LIN {X -6.399,Y 248.174,Z 120.000,A 0.000,B 0.000,C 180.000,E1 0.000} C_DIS
LIN {X -19.159,Y 247.517,Z 120.000,A 0.000,B 0.000,C 180.000,E1 0.000} C_DIS
LIN {X -31.876,Y 246.202,Z 120.000,A 0.000,B 0.000,C 180.000,E1 0.000} C_DIS
LIN {X -44.507,Y 244.235,Z 120.000,A 0.000,B 0.000,C 180.000,E1 0.000} C_DIS
LIN {X -57.020,Y 241.620,Z 120.000,A 0.000,B 0.000,C 180.000,E1 0.000} C_DIS
LIN {X -69.385,Y 238.363,Z 120.000,A 0.000,B 0.000,C 180.000,E1 0.000} C_DIS
LIN {X -81.563,Y 234.476,Z 120.000,A 0.000,B 0.000,C 180.000,E1 0.000} C_DIS
LIN {X -93.525,Y 229.967,Z 120.000,A 0.000,B 0.000,C 180.000,E1 0.000} C_DIS
LIN {X -105.240,Y 224.847,Z 120.000,A 0.000,B 0.000,C 180.000,E1 0.000} C_DIS
LIN {X -116.676,Y 219.131,Z 120.000,A 0.000,B 0.000,C 180.000,E1 0.000} C_DIS
LIN {X -127.801,Y 212.835,Z 120.000,A 0.000,B 0.000,C 180.000,E1 0.000} C_DIS
LIN {X -138.588,Y 205.972,Z 120.000,A 0.000,B 0.000,C 180.000,E1 0.000} C_DIS
LIN {X -149.007,Y 198.566,Z 120.000,A 0.000,B 0.000,C 180.000,E1 0.000} C_DIS
LIN {X -159.031,Y 190.632,Z 120.000,A 0.000,B 0.000,C 180.000,E1 0.000} C_DIS
LIN {X -168.634,Y 182.192,Z 120.000,A 0.000,B 0.000,C 180.000,E1 0.000} C_DIS
LIN {X -177.790,Y 173.268,Z 120.000,A 0.000,B 0.000,C 180.000,E1 0.000} C_DIS
LIN {X -186.475,Y 163.887,Z 120.000,A 0.000,B 0.000,C 180.000,E1 0.000} C_DIS
LIN {X -194.663,Y 154.071,Z 120.000,A 0.000,B 0.000,C 180.000,E1 0.000} C_DIS
LIN {X -202.336,Y 143.846,Z 120.000,A 0.000,B 0.000,C 180.000,E1 0.000} C_DIS
LIN {X -209.473,Y 133.237,Z 120.000,A 0.000,B 0.000,C 180.000,E1 0.000} C_DIS
LIN {X -216.056,Y 122.277,Z 120.000,A 0.000,B 0.000,C 180.000,E1 0.000} C_DIS
LIN {X -222.063,Y 110.995,Z 120.000,A 0.000,B 0.000,C 180.000,E1 0.000} C_DIS
LIN {X -227.482,Y 99.416,Z 120.000,A 0.000,B 0.000,C 180.000,E1 0.000} C_DIS
LIN {X -232.298,Y 87.573,Z 120.000,A 0.000,B 0.000,C 180.000,E1 0.000} C_DIS
LIN {X -236.498,Y 75.499,Z 120.000,A 0.000,B 0.000,C 180.000,E1 0.000} C_DIS
LIN {X -240.071,Y 63.225,Z 120.000,A 0.000,B 0.000,C 180.000,E1 0.000} C_DIS
LIN {X -243.008,Y 50.781,Z 120.000,A 0.000,B 0.000,C 180.000,E1 0.000} C_DIS
LIN {X -245.300,Y 38.205,Z 120.000,A 0.000,B 0.000,C 180.000,E1 0.000} C_DIS
LIN {X -246.940,Y 25.526,Z 120.000,A 0.000,B 0.000,C 180.000,E1 0.000} C_DIS
LIN {X -247.927,Y 12.780,Z 120.000,A 0.000,B 0.000,C 180.000,E1 0.000} C_DIS
LIN {X -248.256,Y 0.000,Z 120.000,A 0.000,B 0.000,C 180.000,E1 0.000} C_DIS
LIN {X -247.927,Y -12.780,Z 120.000,A 0.000,B 0.000,C 180.000,E1 0.000} C_DIS
LIN {X -246.940,Y -25.526,Z 120.000,A 0.000,B 0.000,C 180.000,E1 0.000} C_DIS
LIN {X -245.300,Y -38.205,Z 120.000,A 0.000,B 0.000,C 180.000,E1 0.000} C_DIS
LIN {X -243.008,Y -50.781,Z 120.000,A 0.000,B 0.000,C 180.000,E1 0.000} C_DIS
LIN {X -240.071,Y -63.225,Z 120.000,A 0.000,B 0.000,C 180.000,E1 0.000} C_DIS
LIN {X -236.498,Y -75.499,Z 120.000,A 0.000,B 0.000,C 180.000,E1 0.000} C_DIS
LIN {X -232.298,Y -87.573,Z 120.000,A 0.000,B 0.000,C 180.000,E1 0.000} C_DIS
LIN {X -227.482,Y -99.416,Z 120.000,A 0.000,B 0.000,C 180.000,E1 0.000} C_DIS
LIN {X -222.063,Y -110.995,Z 120.000,A 0.000,B 0.000,C 180.000,E1 0.000} C_DIS
LIN {X -216.056,Y -122.277,Z 120.000,A 0.000,B 0.000,C 180.000,E1 0.000} C_DIS
LIN {X -209.473,Y -133.237,Z 120.000,A 0.000,B 0.000,C 180.000,E1 0.000} C_DIS
LIN {X -202.336,Y -143.846,Z 120.000,A 0.000,B 0.000,C 180.000,E1 0.000} C_DIS
LIN {X -194.663,Y -154.071,Z 120.000,A 0.000,B 0.000,C 180.000,E1 0.000} C_DIS
LIN {X -186.475,Y -163.887,Z 120.000,A 0.000,B 0.000,C 180.000,E1 0.000} C_DIS
LIN {X -177.790,Y -173.268,Z 120.000,A 0.000,B 0.000,C 180.000,E1 0.000} C_DIS
LIN {X -168.634,Y -182.192,Z 120.000,A 0.000,B 0.000,C 180.000,E1 0.000} C_DIS
LIN {X -159.031,Y -190.632,Z 120.000,A 0.000,B 0.000,C 180.000,E1 0.000} C_DIS
LIN {X -149.007,Y -198.566,Z 120.000,A 0.000,B 0.000,C 180.000,E1 0.000} C_DIS
LIN {X -138.588,Y -205.972,Z 120.000,A 0.000,B 0.000,C 180.000,E1 0.000} C_DIS
LIN {X -127.801,Y -212.835,Z 120.000,A 0.000,B 0.000,C 180.000,E1 0.000} C_DIS
LIN {X -116.676,Y -219.131,Z 120.000,A 0.000,B 0.000,C 180.000,E1 0.000} C_DIS
LIN {X -105.240,Y -224.847,Z 120.000,A 0.000,B 0.000,C 180.000,E1 0.000} C_DIS
LIN {X -93.525,Y -229.967,Z 120.000,A 0.000,B 0.000,C 180.000,E1 0.000} C_DIS
LIN {X -81.563,Y -234.476,Z 120.000,A 0.000,B 0.000,C 180.000,E1 0.000} C_DIS
LIN {X -69.385,Y -238.363,Z 120.000,A 0.000,B 0.000,C 180.000,E1 0.000} C_DIS
LIN {X -57.020,Y -241.620,Z 120.000,A 0.000,B 0.000,C 180.000,E1 0.000} C_DIS
LIN {X -44.507,Y -244.235,Z 120.000,A 0.000,B 0.000,C 180.000,E1 0.000} C_DIS
LIN {X -31.876,Y -246.202,Z 120.000,A 0.000,B 0.000,C 180.000,E1 0.000} C_DIS
LIN {X -19.160,Y -247.517,Z 120.000,A 0.000,B 0.000,C 180.000,E1 0.000} C_DIS
LIN {X -6.393,Y -248.174,Z 120.000,A 0.000,B 0.000,C 180.000,E1 0.000} C_DIS
LIN {X 6.399,Y -248.174,Z 120.000,A 0.000,B 0.000,C 180.000,E1 0.000} C_DIS
LIN {X 19.159,Y -247.517,Z 120.000,A 0.000,B 0.000,C 180.000,E1 0.000} C_DIS
LIN {X 31.876,Y -246.202,Z 120.000,A 0.000,B 0.000,C 180.000,E1 0.000} C_DIS
LIN {X 44.507,Y -244.235,Z 120.000,A 0.000,B 0.000,C 180.000,E1 0.000} C_DIS
LIN {X 57.020,Y -241.620,Z 120.000,A 0.000,B 0.000,C 180.000,E1 0.000} C_DIS
LIN {X 69.385,Y -238.363,Z 120.000,A 0.000,B 0.000,C 180.000,E1 0.000} C_DIS
LIN {X 81.563,Y -234.476,Z 120.000,A 0.000,B 0.000,C 180.000,E1 0.000} C_DIS
LIN {X 93.525,Y -229.967,Z 120.000,A 0.000,B 0.000,C 180.000,E1 0.000} C_DIS
LIN {X 105.240,Y -224.847,Z 120.000,A 0.000,B 0.000,C 180.000,E1 0.000} C_DIS
LIN {X 116.676,Y -219.131,Z 120.000,A 0.000,B 0.000,C 180.000,E1 0.000} C_DIS
LIN {X 127.801,Y -212.835,Z 120.000,A 0.000,B 0.000,C 180.000,E1 0.000} C_DIS
LIN {X 138.588,Y -205.972,Z 120.000,A 0.000,B 0.000,C 180.000,E1 0.000} C_DIS
LIN {X 149.007,Y -198.566,Z 120.000,A 0.000,B 0.000,C 180.000,E1 0.000} C_DIS
LIN {X 159.031,Y -190.632,Z 120.000,A 0.000,B 0.000,C 180.000,E1 0.000} C_DIS
LIN {X 168.634,Y -182.192,Z 120.000,A 0.000,B 0.000,C 180.000,E1 0.000} C_DIS
LIN {X 177.790,Y -173.268,Z 120.000,A 0.000,B 0.000,C 180.000,E1 0.000} C_DIS
LIN {X 186.475,Y -163.887,Z 120.000,A 0.000,B 0.000,C 180.000,E1 0.000} C_DIS
LIN {X 194.663,Y -154.071,Z 120.000,A 0.000,B 0.000,C 180.000,E1 0.000} C_DIS
LIN {X 202.336,Y -143.846,Z 120.000,A 0.000,B 0.000,C 180.000,E1 0.000} C_DIS
LIN {X 209.473,Y -133.237,Z 120.000,A 0.000,B 0.000,C 180.000,E1 0.000} C_DIS
LIN {X 216.056,Y -122.277,Z 120.000,A 0.000,B 0.000,C 180.000,E1 0.000} C_DIS
LIN {X 222.063,Y -110.995,Z 120.000,A 0.000,B 0.000,C 180.000,E1 0.000} C_DIS
LIN {X 227.482,Y -99.416,Z 120.000,A 0.000,B 0.000,C 180.000,E1 0.000} C_DIS
LIN {X 232.298,Y -87.573,Z 120.000,A 0.000,B 0.000,C 180.000,E1 0.000} C_DIS
LIN {X 236.498,Y -75.499,Z 120.000,A 0.000,B 0.000,C 180.000,E1 0.000} C_DIS
LIN {X 240.071,Y -63.225,Z 120.000,A 0.000,B 0.000,C 180.000,E1 0.000} C_DIS
LIN {X 243.008,Y -50.781,Z 120.000,A 0.000,B 0.000,C 180.000,E1 0.000} C_DIS
LIN {X 245.300,Y -38.205,Z 120.000,A 0.000,B 0.000,C 180.000,E1 0.000} C_DIS
LIN {X 246.940,Y -25.526,Z 120.000,A 0.000,B 0.000,C 180.000,E1 0.000} C_DIS
LIN {X 247.927,Y -12.780,Z 120.000,A 0.000,B 0.000,C 180.000,E1 0.000} C_DIS
LIN {X 248.256,Y 0.000,Z 120.000,A 0.000,B 0.000,C 180.000,E1 0.000} C_DIS
;rapid-leaky
$VEL.CP=0.3
LIN {X 60.082,Y -222.448,Z 120.000,A 0.000,B 0.000,C 180.000,E1 0.000} C_DIS
;bead-sparse_infill
$VEL.CP=0.67
LIN {X 222.505,Y -60.024,Z 120.000,A 0.000,B 0.000,C 180.000,E1 0.000} C_DIS
LIN {X 222.891,Y -58.700,Z 120.000,A 0.000,B 0.000,C 180.000,E1 0.000} C_DIS
LIN {X 225.618,Y -47.146,Z 120.000,A 0.000,B 0.000,C 180.000,E1 0.000} C_DIS
LIN {X 227.745,Y -35.472,Z 120.000,A 0.000,B 0.000,C 180.000,E1 0.000} C_DIS
LIN {X 229.269,Y -23.700,Z 120.000,A 0.000,B 0.000,C 180.000,E1 0.000} C_DIS
LIN {X 230.185,Y -11.866,Z 120.000,A 0.000,B 0.000,C 180.000,E1 0.000} C_DIS
LIN {X 230.490,Y 0.000,Z 120.000,A 0.000,B 0.000,C 180.000,E1 0.000} C_DIS
LIN {X 230.185,Y 11.866,Z 120.000,A 0.000,B 0.000,C 180.000,E1 0.000} C_DIS
LIN {X 229.269,Y 23.700,Z 120.000,A 0.000,B 0.000,C 180.000,E1 0.000} C_DIS
LIN {X 227.745,Y 35.472,Z 120.000,A 0.000,B 0.000,C 180.000,E1 0.000} C_DIS
LIN {X 225.618,Y 47.146,Z 120.000,A 0.000,B 0.000,C 180.000,E1 0.000} C_DIS
LIN {X 222.891,Y 58.700,Z 120.000,A 0.000,B 0.000,C 180.000,E1 0.000} C_DIS
LIN {X 219.574,Y 70.096,Z 120.000,A 0.000,B 0.000,C 180.000,E1 0.000} C_DIS
LIN {X 215.674,Y 81.306,Z 120.000,A 0.000,B 0.000,C 180.000,E1 0.000} C_DIS
LIN {X 213.125,Y 87.574,Z 120.000,A 0.000,B 0.000,C 180.000,E1 0.000} C_DIS
LIN {X -87.615,Y -213.167,Z 120.000,A 0.000,B 0.000,C 180.000,E1 0.000} C_DIS
LIN {X -97.709,Y -208.756,Z 120.000,A 0.000,B 0.000,C 180.000,E1 0.000} C_DIS
LIN {X -108.326,Y -203.449,Z 120.000,A 0.000,B 0.000,C 180.000,E1 0.000} C_DIS
LIN {X -118.655,Y -197.604,Z 120.000,A 0.000,B 0.000,C 180.000,E1 0.000} C_DIS
LIN {X -128.670,Y -191.232,Z 120.000,A 0.000,B 0.000,C 180.000,E1 0.000} C_DIS
LIN {X -138.344,Y -184.356,Z 120.000,A 0.000,B 0.000,C 180.000,E1 0.000} C_DIS
LIN {X -147.650,Y -176.990,Z 120.000,A 0.000,B 0.000,C 180.000,E1 0.000} C_DIS
LIN {X -156.566,Y -169.154,Z 120.000,A 0.000,B 0.000,C 180.000,E1 0.000} C_DIS
LIN {X -165.067,Y -160.868,Z 120.000,A 0.000,B 0.000,C 180.000,E1 0.000} C_DIS
LIN {X -173.130,Y -152.159,Z 120.000,A 0.000,B 0.000,C 180.000,E1 0.000} C_DIS
LIN {X -177.885,Y -146.459,Z 120.000,A 0.000,B 0.000,C 180.000,E1 0.000} C_DIS
LIN {X 146.486,Y 177.912,Z 120.000,A 0.000,B 0.000,C 180.000,E1 0.000} C_DIS
LIN {X 138.344,Y 184.356,Z 120.000,A 0.000,B 0.000,C 180.000,E1 0.000} C_DIS
LIN {X 128.670,Y 191.232,Z 120.000,A 0.000,B 0.000,C 180.000,E1 0.000} C_DIS
LIN {X 118.655,Y 197.604,Z 120.000,A 0.000,B 0.000,C 180.000,E1 0.000} C_DIS
LIN {X 108.326,Y 203.449,Z 120.000,A 0.000,B 0.000,C 180.000,E1 0.000} C_DIS
LIN {X 97.709,Y 208.756,Z 120.000,A 0.000,B 0.000,C 180.000,E1 0.000} C_DIS
LIN {X 86.832,Y 213.510,Z 120.000,A 0.000,B 0.000,C 180.000,E1 0.000} C_DIS
LIN {X 75.727,Y 217.696,Z 120.000,A 0.000,B 0.000,C 180.000,E1 0.000} C_DIS
LIN {X 64.420,Y 221.305,Z 120.000,A 0.000,B 0.000,C 180.000,E1 0.000} C_DIS
LIN {X 52.939,Y 224.329,Z 120.000,A 0.000,B 0.000,C 180.000,E1 0.000} C_DIS
LIN {X 41.323,Y 226.757,Z 120.000,A 0.000,B 0.000,C 180.000,E1 0.000} C_DIS
LIN {X 38.753,Y 227.157,Z 120.000,A 0.000,B 0.000,C 180.000,E1 0.000} C_DIS
LIN {X -227.149,Y -38.745,Z 120.000,A 0.000,B 0.000,C 180.000,E1 0.000} C_DIS
;rapid-leaky
$VEL.CP=0.3
LIN {X 144.698,Y 215.055,Z 130.000,A 0.000,B 0.000,C 180.000,E1 0.000} C_DIS
;bead-perimeter_outer
$VEL.CP=0.66
LIN {X 133.436,Y 222.219,Z 130.000,A 0.000,B 0.000,C 180.000,E1 0.000} C_DIS
LIN {X 121.819,Y 228.793,Z 130.000,A 0.000,B 0.000,C 180.000,E1 0.000} C_DIS
LIN {X 109.880,Y 234.761,Z 130.000,A 0.000,B 0.000,C 180.000,E1 0.000} C_DIS
LIN {X 97.650,Y 240.106,Z 130.000,A 0.000,B 0.000,C 180.000,E1 0.000} C_DIS
LIN {X 85.159,Y 244.815,Z 130.000,A 0.000,B 0.000,C 180.000,E1 0.000} C_DIS
LIN {X 72.444,Y 248.874,Z 130.000,A 0.000,B 0.000,C 180.000,E1 0.000} C_DIS
LIN {X 59.536,Y 252.273,Z 130.000,A 0.000,B 0.000,C 180.000,E1 0.000} C_DIS
LIN {X 46.470,Y 255.003,Z 130.000,A 0.000,B 0.000,C 180.000,E1 0.000} C_DIS
LIN {X 33.281,Y 257.058,Z 130.000,A 0.000,B 0.000,C 180.000,E1 0.000} C_DIS
LIN {X 20.004,Y 258.430,Z 130.000,A 0.000,B 0.000,C 180.000,E1 0.000} C_DIS
LIN {X 6.674,Y 259.117,Z 130.000,A 0.000,B 0.000,C 180.000,E1 0.000} C_DIS
LIN {X -6.674,Y 259.117,Z 130.000,A 0.000,B 0.000,C 180.000,E1 0.000} C_DIS
LIN {X -20.004,Y 258.430,Z 130.000,A 0.000,B 0.000,C 180.000,E1 0.000} C_DIS
LIN {X -33.281,Y 257.058,Z 130.000,A 0.000,B 0.000,C 180.000,E1 0.000} C_DIS
LIN {X -46.470,Y 255.003,Z 130.000,A 0.000,B 0.000,C 180.000,E1 0.000} C_DIS
LIN {X -59.536,Y 252.273,Z 130.000,A 0.000,B 0.000,C 180.000,E1 0.000} C_DIS
LIN {X -72.444,Y 248.874,Z 130.000,A 0.000,B 0.000,C 180.000,E1 0.000} C_DIS
LIN {X -85.159,Y 244.815,Z 130.000,A 0.000,B 0.000,C 180.000,E1 0.000} C_DIS
LIN {X -97.649,Y 240.106,Z 130.000,A 0.000,B 0.000,C 180.000,E1 0.000} C_DIS
LIN {X -109.880,Y 234.761,Z 130.000,A 0.000,B 0.000,C 180.000,E1 0.000} C_DIS
LIN {X -121.819,Y 228.793,Z 130.000,A 0.000,B 0.000,C 180.000,E1 0.000} C_DIS
LIN {X -133.436,Y 222.219,Z 130.000,A 0.000,B 0.000,C 180.000,E1 0.000} C_DIS
LIN {X -144.698,Y 215.055,Z 130.000,A 0.000,B 0.000,C 180.000,E1 0.000} C_DIS
LIN {X -155.578,Y 207.321,Z 130.000,A 0.000,B 0.000,C 180.000,E1 0.000} C_DIS
LIN {X -166.044,Y 199.038,Z 130.000,A 0.000,B 0.000,C 180.000,E1 0.000} C_DIS
LIN {X -176.069,Y 190.226,Z 130.000,A 0.000,B 0.000,C 180.000,E1 0.000} C_DIS
LIN {X -185.629,Y 180.909,Z 130.000,A 0.000,B 0.000,C 180.000,E1 0.000} C_DIS
LIN {X -194.696,Y 171.114,Z 130.000,A 0.000,B 0.000,C 180.000,E1 0.000} C_DIS
LIN {X -203.246,Y 160.864,Z 130.000,A 0.000,B 0.000,C 180.000,E1 0.000} C_DIS
LIN {X -211.258,Y 150.188,Z 130.000,A 0.000,B 0.000,C 180.000,E1 0.000} C_DIS
LIN {X -218.710,Y 139.113,Z 130.000,A 0.000,B 0.000,C 180.000,E1 0.000} C_DIS
LIN {X -225.581,Y 127.671,Z 130.000,A 0.000,B 0.000,C 180.000,E1 0.000} C_DIS
LIN {X -231.854,Y 115.889,Z 130.000,A 0.000,B 0.000,C 180.000,E1 0.000} C_DIS
LIN {X -237.513,Y 103.799,Z 130.000,A 0.000,B 0.000,C 180.000,E1 0.000} C_DIS
LIN {X -242.541,Y 91.435,Z 130.000,A 0.000,B 0.000,C 180.000,E1 0.000} C_DIS
LIN {X -246.926,Y 78.828,Z 130.000,A 0.000,B 0.000,C 180.000,E1 0.000} C_DIS
LIN {X -250.657,Y 66.011,Z 130.000,A 0.000,B 0.000,C 180.000,E1 0.000} C_DIS
LIN {X -253.722,Y 53.021,Z 130.000,A 0.000,B 0.000,C 180.000,E1 0.000} C_DIS
LIN {X -256.116,Y 39.889,Z 130.000,A 0.000,B 0.000,C 180.000,E1 0.000} C_DIS
LIN {X -257.830,Y 26.652,Z 130.000,A 0.000,B 0.000,C 180.000,E1 0.000} C_DIS
LIN {X -258.859,Y 13.344,Z 130.000,A 0.000,B 0.000,C 180.000,E1 0.000} C_DIS
LIN {X -259.203,Y 0.000,Z 130.000,A 0.000,B 0.000,C 180.000,E1 0.000} C_DIS
LIN {X -258.859,Y -13.344,Z 130.000,A 0.000,B 0.000,C 180.000,E1 0.000} C_DIS
LIN {X -257.830,Y -26.652,Z 130.000,A 0.000,B 0.000,C 180.000,E1 0.000} C_DIS
LIN {X -256.116,Y -39.889,Z 130.000,A 0.000,B 0.000,C 180.000,E1 0.000} C_DIS
LIN {X -253.722,Y -53.021,Z 130.000,A 0.000,B 0.000,C 180.000,E1 0.000} C_DIS
LIN {X -250.657,Y -66.011,Z 130.000,A 0.000,B 0.000,C 180.000,E1 0.000} C_DIS
LIN {X -246.926,Y -78.828,Z 130.000,A 0.000,B 0.000,C 180.000,E1 0.000} C_DIS
LIN {X -242.541,Y -91.435,Z 130.000,A 0.000,B 0.000,C 180.000,E1 0.000} C_DIS
LIN {X -237.513,Y -103.799,Z 130.000,A 0.000,B 0.000,C 180.000,E1 0.000} C_DIS
LIN {X -231.854,Y -115.889,Z 130.000,A 0.000,B 0.000,C 180.000,E1 0.000} C_DIS
LIN {X -225.581,Y -127.671,Z 130.000,A 0.000,B 0.000,C 180.000,E1 0.000} C_DIS
LIN {X -218.710,Y -139.113,Z 130.000,A 0.000,B 0.000,C 180.000,E1 0.000} C_DIS
LIN {X -211.258,Y -150.188,Z 130.000,A 0.000,B 0.000,C 180.000,E1 0.000} C_DIS
LIN {X -203.246,Y -160.864,Z 130.000,A 0.000,B 0.000,C 180.000,E1 0.000} C_DIS
LIN {X -194.696,Y -171.114,Z 130.000,A 0.000,B 0.000,C 180.000,E1 0.000} C_DIS
LIN {X -185.629,Y -180.909,Z 130.000,A 0.000,B 0.000,C 180.000,E1 0.000} C_DIS
LIN {X -176.069,Y -190.226,Z 130.000,A 0.000,B 0.000,C 180.000,E1 0.000} C_DIS
LIN {X -166.044,Y -199.038,Z 130.000,A 0.000,B 0.000,C 180.000,E1 0.000} C_DIS
LIN {X -155.578,Y -207.321,Z 130.000,A 0.000,B 0.000,C 180.000,E1 0.000} C_DIS
LIN {X -144.698,Y -215.055,Z 130.000,A 0.000,B 0.000,C 180.000,E1 0.000} C_DIS
LIN {X -133.436,Y -222.219,Z 130.000,A 0.000,B 0.000,C 180.000,E1 0.000} C_DIS
LIN {X -121.819,Y -228.793,Z 130.000,A 0.000,B 0.000,C 180.000,E1 0.000} C_DIS
LIN {X -109.880,Y -234.761,Z 130.000,A 0.000,B 0.000,C 180.000,E1 0.000} C_DIS
LIN {X -97.650,Y -240.106,Z 130.000,A 0.000,B 0.000,C 180.000,E1 0.000} C_DIS
LIN {X -85.159,Y -244.815,Z 130.000,A 0.000,B 0.000,C 180.000,E1 0.000} C_DIS
LIN {X -72.444,Y -248.874,Z 130.000,A 0.000,B 0.000,C 180.000,E1 0.000} C_DIS
LIN {X -59.536,Y -252.273,Z 130.000,A 0.000,B 0.000,C 180.000,E1 0.000} C_DIS
LIN {X -46.470,Y -255.003,Z 130.000,A 0.000,B 0.000,C 180.000,E1 0.000} C_DIS
LIN {X -33.281,Y -257.058,Z 130.000,A 0.000,B 0.000,C 180.000,E1 0.000} C_DIS
LIN {X -20.004,Y -258.430,Z 130.000,A 0.000,B 0.000,C 180.000,E1 0.000} C_DIS
LIN {X -6.674,Y -259.117,Z 130.000,A 0.000,B 0.000,C 180.000,E1 0.000} C_DIS
LIN {X 6.674,Y -259.117,Z 130.000,A 0.000,B 0.000,C 180.000,E1 0.000} C_DIS
LIN {X 20.004,Y -258.430,Z 130.000,A 0.000,B 0.000,C 180.000,E1 0.000} C_DIS
LIN {X 33.281,Y -257.058,Z 130.000,A 0.000,B 0.000,C 180.000,E1 0.000} C_DIS
LIN {X 46.470,Y -255.003,Z 130.000,A 0.000,B 0.000,C 180.000,E1 0.000} C_DIS
LIN {X 59.536,Y -252.273,Z 130.000,A 0.000,B 0.000,C 180.000,E1 0.000} C_DIS
LIN {X 72.444,Y -248.874,Z 130.000,A 0.000,B 0.000,C 180.000,E1 0.000} C_DIS
LIN {X 85.159,Y -244.815,Z 130.000,A 0.000,B 0.000,C 180.000,E1 0.000} C_DIS
LIN {X 97.649,Y -240.106,Z 130.000,A 0.000,B 0.000,C 180.000,E1 0.000} C_DIS
LIN {X 109.880,Y -234.761,Z 130.000,A 0.000,B 0.000,C 180.000,E1 0.000} C_DIS
LIN {X 121.819,Y -228.793,Z 130.000,A 0.000,B 0.000,C 180.000,E1 0.000} C_DIS
LIN {X 133.436,Y -222.219,Z 130.000,A 0.000,B 0.000,C 180.000,E1 0.000} C_DIS
LIN {X 144.698,Y -215.055,Z 130.000,A 0.000,B 0.000,C 180.000,E1 0.000} C_DIS
LIN {X 155.578,Y -207.321,Z 130.000,A 0.000,B 0.000,C 180.000,E1 0.000} C_DIS
LIN {X 166.044,Y -199.038,Z 130.000,A 0.000,B 0.000,C 180.000,E1 0.000} C_DIS
LIN {X 176.069,Y -190.226,Z 130.000,A 0.000,B 0.000,C 180.000,E1 0.000} C_DIS
LIN {X 185.629,Y -180.909,Z 130.000,A 0.000,B 0.000,C 180.000,E1 0.000} C_DIS
LIN {X 194.696,Y -171.114,Z 130.000,A 0.000,B 0.000,C 180.000,E1 0.000} C_DIS
LIN {X 203.246,Y -160.864,Z 130.000,A 0.000,B 0.000,C 180.000,E1 0.000} C_DIS
LIN {X 211.258,Y -150.188,Z 130.000,A 0.000,B 0.000,C 180.000,E1 0.000} C_DIS
LIN {X 218.710,Y -139.113,Z 130.000,A 0.000,B 0.000,C 180.000,E1 0.000} C_DIS
LIN {X 225.581,Y -127.671,Z 130.000,A 0.000,B 0.000,C 180.000,E1 0.000} C_DIS
LIN {X 231.854,Y -115.889,Z 130.000,A 0.000,B 0.000,C 180.000,E1 0.000} C_DIS
LIN {X 237.513,Y -103.799,Z 130.000,A 0.000,B 0.000,C 180.000,E1 0.000} C_DIS
LIN {X 242.541,Y -91.435,Z 130.000,A 0.000,B 0.000,C 180.000,E1 0.000} C_DIS
LIN {X 246.926,Y -78.828,Z 130.000,A 0.000,B 0.000,C 180.000,E1 0.000} C_DIS
LIN {X 250.657,Y -66.011,Z 130.000,A 0.000,B 0.000,C 180.000,E1 0.000} C_DIS
LIN {X 253.722,Y -53.021,Z 130.000,A 0.000,B 0.000,C 180.000,E1 0.000} C_DIS
LIN {X 256.116,Y -39.889,Z 130.000,A 0.000,B 0.000,C 180.000,E1 0.000} C_DIS
LIN {X 257.830,Y -26.652,Z 130.000,A 0.000,B 0.000,C 180.000,E1 0.000} C_DIS
LIN {X 258.859,Y -13.344,Z 130.000,A 0.000,B 0.000,C 180.000,E1 0.000} C_DIS
LIN {X 259.203,Y 0.000,Z 130.000,A 0.000,B 0.000,C 180.000,E1 0.000} C_DIS
LIN {X 258.859,Y 13.344,Z 130.000,A 0.000,B 0.000,C 180.000,E1 0.000} C_DIS
LIN {X 257.830,Y 26.652,Z 130.000,A 0.000,B 0.000,C 180.000,E1 0.000} C_DIS
LIN {X 256.116,Y 39.889,Z 130.000,A 0.000,B 0.000,C 180.000,E1 0.000} C_DIS
LIN {X 253.722,Y 53.021,Z 130.000,A 0.000,B 0.000,C 180.000,E1 0.000} C_DIS
LIN {X 250.657,Y 66.011,Z 130.000,A 0.000,B 0.000,C 180.000,E1 0.000} C_DIS
LIN {X 246.926,Y 78.828,Z 130.000,A 0.000,B 0.000,C 180.000,E1 0.000} C_DIS
LIN {X 242.541,Y 91.435,Z 130.000,A 0.000,B 0.000,C 180.000,E1 0.000} C_DIS
LIN {X 237.513,Y 103.799,Z 130.000,A 0.000,B 0.000,C 180.000,E1 0.000} C_DIS
LIN {X 231.854,Y 115.889,Z 130.000,A 0.000,B 0.000,C 180.000,E1 0.000} C_DIS
LIN {X 225.581,Y 127.671,Z 130.000,A 0.000,B 0.000,C 180.000,E1 0.000} C_DIS
LIN {X 218.710,Y 139.113,Z 130.000,A 0.000,B 0.000,C 180.000,E1 0.000} C_DIS
LIN {X 211.258,Y 150.188,Z 130.000,A 0.000,B 0.000,C 180.000,E1 0.000} C_DIS
LIN {X 203.246,Y 160.864,Z 130.000,A 0.000,B 0.000,C 180.000,E1 0.000} C_DIS
LIN {X 194.696,Y 171.114,Z 130.000,A 0.000,B 0.000,C 180.000,E1 0.000} C_DIS
LIN {X 185.629,Y 180.909,Z 130.000,A 0.000,B 0.000,C 180.000,E1 0.000} C_DIS
LIN {X 176.069,Y 190.226,Z 130.000,A 0.000,B 0.000,C 180.000,E1 0.000} C_DIS
LIN {X 166.044,Y 199.038,Z 130.000,A 0.000,B 0.000,C 180.000,E1 0.000} C_DIS
LIN {X 155.578,Y 207.321,Z 130.000,A 0.000,B 0.000,C 180.000,E1 0.000} C_DIS
LIN {X 144.698,Y 215.055,Z 130.000,A 0.000,B 0.000,C 180.000,E1 0.000} C_DIS
;rapid-leaky
$VEL.CP=0.3
LIN {X 136.020,Y 202.157,Z 130.000,A 0.000,B 0.000,C 180.000,E1 0.000} C_DIS
;bead-perimeter_inner
$VEL.CP=0.66
LIN {X 125.433,Y 208.892,Z 130.000,A 0.000,B 0.000,C 180.000,E1 0.000} C_DIS
LIN {X 114.513,Y 215.072,Z 130.000,A 0.000,B 0.000,C 180.000,E1 0.000} C_DIS
LIN {X 103.290,Y 220.682,Z 130.000,A 0.000,B 0.000,C 180.000,E1 0.000} C_DIS
LIN {X 91.794,Y 225.706,Z 130.000,A 0.000,B 0.000,C 180.000,E1 0.000} C_DIS
LIN {X 80.052,Y 230.132,Z 130.000,A 0.000,B 0.000,C 180.000,E1 0.000} C_DIS
LIN {X 68.099,Y 233.948,Z 130.000,A 0.000,B 0.000,C 180.000,E1 0.000} C_DIS
LIN {X 55.965,Y 237.144,Z 130.000,A 0.000,B 0.000,C 180.000,E1 0.000} C_DIS
LIN {X 43.683,Y 239.710,Z 130.000,A 0.000,B 0.000,C 180.000,E1 0.000} C_DIS
LIN {X 31.285,Y 241.642,Z 130.000,A 0.000,B 0.000,C 180.000,E1 0.000} C_DIS
LIN {X 18.805,Y 242.932,Z 130.000,A 0.000,B 0.000,C 180.000,E1 0.000} C_DIS
LIN {X 6.274,Y 243.577,Z 130.000,A 0.000,B 0.000,C 180.000,E1 0.000} C_DIS
LIN {X -6.274,Y 243.577,Z 130.000,A 0.000,B 0.000,C 180.000,E1 0.000} C_DIS
LIN {X -18.805,Y 242.932,Z 130.000,A 0.000,B 0.000,C 180.000,E1 0.000} C_DIS
LIN {X -31.285,Y 241.642,Z 130.000,A 0.000,B 0.000,C 180.000,E1 0.000} C_DIS
LIN {X -43.683,Y 239.710,Z 130.000,A 0.000,B 0.000,C 180.000,E1 0.000} C_DIS
LIN {X -55.965,Y 237.144,Z 130.000,A 0.000,B 0.000,C 180.000,E1 0.000} C_DIS
LIN {X -68.099,Y 233.948,Z 130.000,A 0.000,B 0.000,C 180.000,E1 0.000} C_DIS
LIN {X -80.052,Y 230.132,Z 130.000,A 0.000,B 0.000,C 180.000,E1 0.000} C_DIS
LIN {X -91.793,Y 225.706,Z 130.000,A 0.000,B 0.000,C 180.000,E1 0.000} C_DIS
LIN {X -103.290,Y 220.682,Z 130.000,A 0.000,B 0.000,C 180.000,E1 0.000} C_DIS
LIN {X -114.513,Y 215.072,Z 130.000,A 0.000,B 0.000,C 180.000,E1 0.000} C_DIS
LIN {X -125.433,Y 208.892,Z 130.000,A 0.000,B 0.000,C 180.000,E1 0.000} C_DIS
LIN {X -136.020,Y 202.157,Z 130.000,A 0.000,B 0.000,C 180.000,E1 0.000} C_DIS
LIN {X -146.248,Y 194.887,Z 130.000,A 0.000,B 0.000,C 180.000,E1 0.000} C_DIS
LIN {X -156.086,Y 187.101,Z 130.000,A 0.000,B 0.000,C 180.000,E1 0.000} C_DIS
LIN {X -165.510,Y 178.818,Z 130.000,A 0.000,B 0.000,C 180.000,E1 0.000} C_DIS
LIN {X -174.496,Y 170.060,Z 130.000,A 0.000,B 0.000,C 180.000,E1 0.000} C_DIS
LIN {X -183.019,Y 160.852,Z 130.000,A 0.000,B 0.000,C 180.000,E1 0.000} C_DIS
LIN {X -191.057,Y 151.216,Z 130.000,A 0.000,B 0.000,C 180.000,E1 0.000} C_DIS
LIN {X -198.589,Y 141.181,Z 130.000,A 0.000,B 0.000,C 180.000,E1 0.000} C_DIS
LIN {X -205.593,Y 130.770,Z 130.000,A 0.000,B 0.000,C 180.000,E1 0.000} C_DIS
LIN {X -212.052,Y 120.015,Z 130.000,A 0.000,B 0.000,C 180.000,E1 0.000} C_DIS
LIN {X -217.949,Y 108.938,Z 130.000,A 0.000,B 0.000,C 180.000,E1 0.000} C_DIS
LIN {X -223.268,Y 97.574,Z 130.000,A 0.000,B 0.000,C 180.000,E1 0.000} C_DIS
LIN {X -227.995,Y 85.952,Z 130.000,A 0.000,B 0.000,C 180.000,E1 0.000} C_DIS
LIN {X -232.117,Y 74.101,Z 130.000,A 0.000,B 0.000,C 180.000,E1 0.000} C_DIS
LIN {X -235.625,Y 62.053,Z 130.000,A 0.000,B 0.000,C 180.000,E1 0.000} C_DIS
LIN {X -238.506,Y 49.841,Z 130.000,A 0.000,B 0.000,C 180.000,E1 0.000} C_DIS
LIN {X -240.756,Y 37.496,Z 130.000,A 0.000,B 0.000,C 180.000,E1 0.000} C_DIS
LIN {X -242.367,Y 25.053,Z 130.000,A 0.000,B 0.000,C 180.000,E1 0.000} C_DIS
LIN {X -243.335,Y 12.544,Z 130.000,A 0.000,B 0.000,C 180.000,E1 0.000} C_DIS
LIN {X -243.658,Y 0.000,Z 130.000,A 0.000,B 0.000,C 180.000,E1 0.000} C_DIS
LIN {X -243.335,Y -12.544,Z 130.000,A 0.000,B 0.000,C 180.000,E1 0.000} C_DIS
LIN {X -242.367,Y -25.053,Z 130.000,A 0.000,B 0.000,C 180.000,E1 0.000} C_DIS
LIN {X -240.756,Y -37.496,Z 130.000,A 0.000,B 0.000,C 180.000,E1 0.000} C_DIS
LIN {X -238.506,Y -49.841,Z 130.000,A 0.000,B 0.000,C 180.000,E1 0.000} C_DIS
LIN {X -235.625,Y -62.053,Z 130.000,A 0.000,B 0.000,C 180.000,E1 0.000} C_DIS
LIN {X -232.117,Y -74.101,Z 130.000,A 0.000,B 0.000,C 180.000,E1 0.000} C_DIS
LIN {X -227.995,Y -85.952,Z 130.000,A 0.000,B 0.000,C 180.000,E1 0.000} C_DIS
LIN {X -223.268,Y -97.574,Z 130.000,A 0.000,B 0.000,C 180.000,E1 0.000} C_DIS
LIN {X -217.949,Y -108.938,Z 130.000,A 0.000,B 0.000,C 180.000,E1 0.000} C_DIS
LIN {X -212.052,Y -120.014,Z 130.000,A 0.000,B 0.000,C 180.000,E1 0.000} C_DIS
LIN {X -205.593,Y -130.770,Z 130.000,A 0.000,B 0.000,C 180.000,E1 0.000} C_DIS
LIN {X -198.589,Y -141.181,Z 130.000,A 0.000,B 0.000,C 180.000,E1 0.000} C_DIS
LIN {X -191.057,Y -151.216,Z 130.000,A 0.000,B 0.000,C 180.000,E1 0.000} C_DIS
LIN {X -183.019,Y -160.852,Z 130.000,A 0.000,B 0.000,C 180.000,E1 0.000} C_DIS
LIN {X -174.496,Y -170.060,Z 130.000,A 0.000,B 0.000,C 180.000,E1 0.000} C_DIS
LIN {X -165.510,Y -178.818,Z 130.000,A 0.000,B 0.000,C 180.000,E1 0.000} C_DIS
LIN {X -156.086,Y -187.101,Z 130.000,A 0.000,B 0.000,C 180.000,E1 0.000} C_DIS
LIN {X -146.248,Y -194.887,Z 130.000,A 0.000,B 0.000,C 180.000,E1 0.000} C_DIS
LIN {X -136.020,Y -202.157,Z 130.000,A 0.000,B 0.000,C 180.000,E1 0.000} C_DIS
LIN {X -125.433,Y -208.892,Z 130.000,A 0.000,B 0.000,C 180.000,E1 0.000} C_DIS
LIN {X -114.513,Y -215.072,Z 130.000,A 0.000,B 0.000,C 180.000,E1 0.000} C_DIS
LIN {X -103.290,Y -220.682,Z 130.000,A 0.000,B 0.000,C 180.000,E1 0.000} C_DIS
LIN {X -91.794,Y -225.706,Z 130.000,A 0.000,B 0.000,C 180.000,E1 0.000} C_DIS
LIN {X -80.052,Y -230.132,Z 130.000,A 0.000,B 0.000,C 180.000,E1 0.000} C_DIS
LIN {X -68.099,Y -233.948,Z 130.000,A 0.000,B 0.000,C 180.000,E1 0.000} C_DIS
LIN {X -55.965,Y -237.144,Z 130.000,A 0.000,B 0.000,C 180.000,E1 0.000} C_DIS
LIN {X -43.683,Y -239.710,Z 130.000,A 0.000,B 0.000,C 180.000,E1 0.000} C_DIS
LIN {X -31.285,Y -241.642,Z 130.000,A 0.000,B 0.000,C 180.000,E1 0.000} C_DIS
LIN {X -18.805,Y -242.932,Z 130.000,A 0.000,B 0.000,C 180.000,E1 0.000} C_DIS
LIN {X -6.274,Y -243.577,Z 130.000,A 0.000,B 0.000,C 180.000,E1 0.000} C_DIS
LIN {X 6.274,Y -243.577,Z 130.000,A 0.000,B 0.000,C 180.000,E1 0.000} C_DIS
LIN {X 18.805,Y -242.932,Z 130.000,A 0.000,B 0.000,C 180.000,E1 0.000} C_DIS
LIN {X 31.285,Y -241.642,Z 130.000,A 0.000,B 0.000,C 180.000,E1 0.000} C_DIS
LIN {X 43.683,Y -239.710,Z 130.000,A 0.000,B 0.000,C 180.000,E1 0.000} C_DIS
LIN {X 55.965,Y -237.144,Z 130.000,A 0.000,B 0.000,C 180.000,E1 0.000} C_DIS
LIN {X 68.099,Y -233.948,Z 130.000,A 0.000,B 0.000,C 180.000,E1 0.000} C_DIS
LIN {X 80.052,Y -230.132,Z 130.000,A 0.000,B 0.000,C 180.000,E1 0.000} C_DIS
LIN {X 91.793,Y -225.706,Z 130.000,A 0.000,B 0.000,C 180.000,E1 0.000} C_DIS
LIN {X 103.290,Y -220.682,Z 130.000,A 0.000,B 0.000,C 180.000,E1 0.000} C_DIS
LIN {X 114.513,Y -215.072,Z 130.000,A 0.000,B 0.000,C 180.000,E1 0.000} C_DIS
LIN {X 125.433,Y -208.892,Z 130.000,A 0.000,B 0.000,C 180.000,E1 0.000} C_DIS
LIN {X 136.020,Y -202.157,Z 130.000,A 0.000,B 0.000,C 180.000,E1 0.000} C_DIS
LIN {X 146.248,Y -194.887,Z 130.000,A 0.000,B 0.000,C 180.000,E1 0.000} C_DIS
LIN {X 156.086,Y -187.101,Z 130.000,A 0.000,B 0.000,C 180.000,E1 0.000} C_DIS
LIN {X 165.510,Y -178.818,Z 130.000,A 0.000,B 0.000,C 180.000,E1 0.000} C_DIS
LIN {X 174.496,Y -170.060,Z 130.000,A 0.000,B 0.000,C 180.000,E1 0.000} C_DIS
LIN {X 183.019,Y -160.852,Z 130.000,A 0.000,B 0.000,C 180.000,E1 0.000} C_DIS
LIN {X 191.057,Y -151.216,Z 130.000,A 0.000,B 0.000,C 180.000,E1 0.000} C_DIS
LIN {X 198.589,Y -141.181,Z 130.000,A 0.000,B 0.000,C 180.000,E1 0.000} C_DIS
LIN {X 205.593,Y -130.770,Z 130.000,A 0.000,B 0.000,C 180.000,E1 0.000} C_DIS
LIN {X 212.052,Y -120.015,Z 130.000,A 0.000,B 0.000,C 180.000,E1 0.000} C_DIS
LIN {X 217.949,Y -108.938,Z 130.000,A 0.000,B 0.000,C 180.000,E1 0.000} C_DIS
LIN {X 223.268,Y -97.574,Z 130.000,A 0.000,B 0.000,C 180.000,E1 0.000} C_DIS
LIN {X 227.995,Y -85.952,Z 130.000,A 0.000,B 0.000,C 180.000,E1 0.000} C_DIS
LIN {X 232.117,Y -74.101,Z 130.000,A 0.000,B 0.000,C 180.000,E1 0.000} C_DIS
LIN {X 235.625,Y -62.053,Z 130.000,A 0.000,B 0.000,C 180.000,E1 0.000} C_DIS
LIN {X 238.506,Y -49.841,Z 130.000,A 0.000,B 0.000,C 180.000,E1 0.000} C_DIS
LIN {X 240.756,Y -37.496,Z 130.000,A 0.000,B 0.000,C 180.000,E1 0.000} C_DIS
LIN {X 242.367,Y -25.053,Z 130.000,A 0.000,B 0.000,C 180.000,E1 0.000} C_DIS
LIN {X 243.335,Y -12.544,Z 130.000,A 0.000,B 0.000,C 180.000,E1 0.000} C_DIS
LIN {X 243.658,Y 0.000,Z 130.000,A 0.000,B 0.000,C 180.000,E1 0.000} C_DIS
LIN {X 243.335,Y 12.544,Z 130.000,A 0.000,B 0.000,C 180.000,E1 0.000} C_DIS
LIN {X 242.367,Y 25.053,Z 130.000,A 0.000,B 0.000,C 180.000,E1 0.000} C_DIS
LIN {X 240.756,Y 37.496,Z 130.000,A 0.000,B 0.000,C 180.000,E1 0.000} C_DIS
LIN {X 238.506,Y 49.841,Z 130.000,A 0.000,B 0.000,C 180.000,E1 0.000} C_DIS
LIN {X 235.625,Y 62.053,Z 130.000,A 0.000,B 0.000,C 180.000,E1 0.000} C_DIS
LIN {X 232.117,Y 74.101,Z 130.000,A 0.000,B 0.000,C 180.000,E1 0.000} C_DIS
LIN {X 227.995,Y 85.952,Z 130.000,A 0.000,B 0.000,C 180.000,E1 0.000} C_DIS
LIN {X 223.268,Y 97.574,Z 130.000,A 0.000,B 0.000,C 180.000,E1 0.000} C_DIS
LIN {X 217.949,Y 108.938,Z 130.000,A 0.000,B 0.000,C 180.000,E1 0.000} C_DIS
LIN {X 212.052,Y 120.014,Z 130.000,A 0.000,B 0.000,C 180.000,E1 0.000} C_DIS
LIN {X 205.593,Y 130.770,Z 130.000,A 0.000,B 0.000,C 180.000,E1 0.000} C_DIS
LIN {X 198.589,Y 141.181,Z 130.000,A 0.000,B 0.000,C 180.000,E1 0.000} C_DIS
LIN {X 191.057,Y 151.216,Z 130.000,A 0.000,B 0.000,C 180.000,E1 0.000} C_DIS
LIN {X 183.019,Y 160.852,Z 130.000,A 0.000,B 0.000,C 180.000,E1 0.000} C_DIS
LIN {X 174.496,Y 170.060,Z 130.000,A 0.000,B 0.000,C 180.000,E1 0.000} C_DIS
LIN {X 165.510,Y 178.818,Z 130.000,A 0.000,B 0.000,C 180.000,E1 0.000} C_DIS
LIN {X 156.086,Y 187.101,Z 130.000,A 0.000,B 0.000,C 180.000,E1 0.000} C_DIS
LIN {X 146.248,Y 194.887,Z 130.000,A 0.000,B 0.000,C 180.000,E1 0.000} C_DIS
LIN {X 136.020,Y 202.157,Z 130.000,A 0.000,B 0.000,C 180.000,E1 0.000} C_DIS
;rapid-leaky
$VEL.CP=0.3
LIN {X 66.814,Y 215.715,Z 130.000,A 0.000,B 0.000,C 180.000,E1 0.000} C_DIS
;bead-sparse_infill
$VEL.CP=0.66
LIN {X 215.752,Y 66.778,Z 130.000,A 0.000,B 0.000,C 180.000,E1 0.000} C_DIS
LIN {X 218.444,Y 57.529,Z 130.000,A 0.000,B 0.000,C 180.000,E1 0.000} C_DIS
LIN {X 221.115,Y 46.208,Z 130.000,A 0.000,B 0.000,C 180.000,E1 0.000} C_DIS
LIN {X 223.202,Y 34.761,Z 130.000,A 0.000,B 0.000,C 180.000,E1 0.000} C_DIS
LIN {X 224.696,Y 23.227,Z 130.000,A 0.000,B 0.000,C 180.000,E1 0.000} C_DIS
LIN {X 225.592,Y 11.630,Z 130.000,A 0.000,B 0.000,C 180.000,E1 0.000} C_DIS
LIN {X 225.892,Y 0.000,Z 130.000,A 0.000,B 0.000,C 180.000,E1 0.000} C_DIS
LIN {X 225.592,Y -11.630,Z 130.000,A 0.000,B 0.000,C 180.000,E1 0.000} C_DIS
LIN {X 224.696,Y -23.227,Z 130.000,A 0.000,B 0.000,C 180.000,E1 0.000} C_DIS
LIN {X 223.202,Y -34.761,Z 130.000,A 0.000,B 0.000,C 180.000,E1 0.000} C_DIS
LIN {X 221.115,Y -46.208,Z 130.000,A 0.000,B 0.000,C 180.000,E1 0.000} C_DIS
LIN {X 218.444,Y -57.529,Z 130.000,A 0.000,B 0.000,C 180.000,E1 0.000} C_DIS
LIN {X 215.193,Y -68.698,Z 130.000,A 0.000,B 0.000,C 180.000,E1 0.000} C_DIS
LIN {X 211.371,Y -79.685,Z 130.000,A 0.000,B 0.000,C 180.000,E1 0.000} C_DIS
LIN {X 209.598,Y -84.046,Z 130.000,A 0.000,B 0.000,C 180.000,E1 0.000} C_DIS
LIN {X -84.082,Y 209.633,Z 130.000,A 0.000,B 0.000,C 180.000,E1 0.000} C_DIS
LIN {X -85.100,Y 209.249,Z 130.000,A 0.000,B 0.000,C 180.000,E1 0.000} C_DIS
LIN {X -95.759,Y 204.592,Z 130.000,A 0.000,B 0.000,C 180.000,E1 0.000} C_DIS
LIN {X -106.163,Y 199.390,Z 130.000,A 0.000,B 0.000,C 180.000,E1 0.000} C_DIS
LIN {X -116.287,Y 193.661,Z 130.000,A 0.000,B 0.000,C 180.000,E1 0.000} C_DIS
LIN {X -126.103,Y 187.417,Z 130.000,A 0.000,B 0.000,C 180.000,E1 0.000} C_DIS
LIN {X -135.585,Y 180.676,Z 130.000,A 0.000,B 0.000,C 180.000,E1 0.000} C_DIS
LIN {X -144.706,Y 173.458,Z 130.000,A 0.000,B 0.000,C 180.000,E1 0.000} C_DIS
LIN {X -153.442,Y 165.780,Z 130.000,A 0.000,B 0.000,C 180.000,E1 0.000} C_DIS
LIN {X -161.773,Y 157.660,Z 130.000,A 0.000,B 0.000,C 180.000,E1 0.000} C_DIS
LIN {X -169.675,Y 149.124,Z 130.000,A 0.000,B 0.000,C 180.000,E1 0.000} C_DIS
LIN {X -174.621,Y 143.195,Z 130.000,A 0.000,B 0.000,C 180.000,E1 0.000} C_DIS
LIN {X 143.214,Y -174.639,Z 130.000,A 0.000,B 0.000,C 180.000,E1 0.000} C_DIS
LIN {X 135.585,Y -180.676,Z 130.000,A 0.000,B 0.000,C 180.000,E1 0.000} C_DIS
LIN {X 126.103,Y -187.417,Z 130.000,A 0.000,B 0.000,C 180.000,E1 0.000} C_DIS
LIN {X 116.287,Y -193.661,Z 130.000,A 0.000,B 0.000,C 180.000,E1 0.000} C_DIS
LIN {X 106.163,Y -199.390,Z 130.000,A 0.000,B 0.000,C 180.000,E1 0.000} C_DIS
LIN {X 95.759,Y -204.592,Z 130.000,A 0.000,B 0.000,C 180.000,E1 0.000} C_DIS
LIN {X 85.100,Y -209.249,Z 130.000,A 0.000,B 0.000,C 180.000,E1 0.000} C_DIS
LIN {X 74.215,Y -213.353,Z 130.000,A 0.000,B 0.000,C 180.000,E1 0.000} C_DIS
LIN {X 63.134,Y -216.890,Z 130.000,A 0.000,B 0.000,C 180.000,E1 0.000} C_DIS
LIN {X 51.885,Y -219.853,Z 130.000,A 0.000,B 0.000,C 180.000,E1 0.000} C_DIS
LIN {X 40.497,Y -222.232,Z 130.000,A 0.000,B 0.000,C 180.000,E1 0.000} C_DIS
LIN {X 34.728,Y -223.131,Z 130.000,A 0.000,B 0.000,C 180.000,E1 0.000} C_DIS
LIN {X -223.196,Y 34.792,Z 130.000,A 0.000,B 0.000,C 180.000,E1 0.000} C_DIS
;rapid-leaky
$VEL.CP=0.3
LIN {X 252.773,Y 26.129,Z 140.000,A 0.000,B 0.000,C 180.000,E1 0.000} C_DIS
;bead-perimeter_outer
$VEL.CP=0.65
LIN {X 251.093,Y 39.106,Z 140.000,A 0.000,B 0.000,C 180.000,E1 0.000} C_DIS
LIN {X 248.746,Y 51.981,Z 140.000,A 0.000,B 0.000,C 180.000,E1 0.000} C_DIS
LIN {X 245.740,Y 64.716,Z 140.000,A 0.000,B 0.000,C 180.000,E1 0.000} C_DIS
LIN {X 242.083,Y 77.282,Z 140.000,A 0.000,B 0.000,C 180.000,E1 0.000} C_DIS
LIN {X 237.784,Y 89.641,Z 140.000,A 0.000,B 0.000,C 180.000,E1 0.000} C_DIS
LIN {X 232.855,Y 101.763,Z 140.000,A 0.000,B 0.000,C 180.000,E1 0.000} C_DIS
LIN {X 227.307,Y 113.614,Z 140.000,A 0.000,B 0.000,C 180.000,E1 0.000} C_DIS
LIN {X 221.157,Y 125.166,Z 140.000,A 0.000,B 0.000,C 180.000,E1 0.000} C_DIS
LIN {X 214.420,Y 136.385,Z 140.000,A 0.000,B 0.000,C 180.000,E1 0.000} C_DIS
LIN {X 207.114,Y 147.242,Z 140.000,A 0.000,B 0.000,C 180.000,E1 0.000} C_DIS
LIN {X 199.260,Y 157.709,Z 140.000,A 0.000,B 0.000,C 180.000,E1 0.000} C_DIS
LIN {X 190.878,Y 167.758,Z 140.000,A 0.000,B 0.000,C 180.000,E1 0.000} C_DIS
LIN {X 181.988,Y 177.361,Z 140.000,A 0.000,B 0.000,C 180.000,E1 0.000} C_DIS
LIN {X 172.616,Y 186.495,Z 140.000,A 0.000,B 0.000,C 180.000,E1 0.000} C_DIS
LIN {X 162.787,Y 195.133,Z 140.000,A 0.000,B 0.000,C 180.000,E1 0.000} C_DIS
LIN {X 152.526,Y 203.255,Z 140.000,A 0.000,B 0.000,C 180.000,E1 0.000} C_DIS
LIN {X 141.860,Y 210.838,Z 140.000,A 0.000,B 0.000,C 180.000,E1 0.000} C_DIS
LIN {X 130.819,Y 217.861,Z 140.000,A 0.000,B 0.000,C 180.000,E1 0.000} C_DIS
LIN {X 119.431,Y 224.306,Z 140.000,A 0.000,B 0.000,C 180.000,E1 0.000} C_DIS
LIN {X 107.725,Y 230.156,Z 140.000,A 0.000,B 0.000,C 180.000,E1 0.000} C_DIS
LIN {X 95.734,Y 235.396,Z 140.000,A 0.000,B 0.000,C 180.000,E1 0.000} C_DIS
LIN {X 83.489,Y 240.013,Z 140.000,A 0.000,B 0.000,C 180.000,E1 0.000} C_DIS
LIN {X 71.023,Y 243.993,Z 140.000,A 0.000,B 0.000,C 180.000,E1 0.000} C_DIS
LIN {X 58.368,Y 247.325,Z 140.000,A 0.000,B 0.000,C 180.000,E1 0.000} C_DIS
LIN {X 45.558,Y 250.002,Z 140.000,A 0.000,B 0.000,C 180.000,E1 0.000} C_DIS
LIN {X 32.628,Y 252.016,Z 140.000,A 0.000,B 0.000,C 180.000,E1 0.000} C_DIS
LIN {X 19.612,Y 253.361,Z 140.000,A 0.000,B 0.000,C 180.000,E1 0.000} C_DIS
LIN {X 6.543,Y 254.035,Z 140.000,A 0.000,B 0.000,C 180.000,E1 0.000} C_DIS
LIN {X -6.543,Y 254.035,Z 140.000,A 0.000,B 0.000,C 180.000,E1 0.000} C_DIS
LIN {X -19.612,Y 253.361,Z 140.000,A 0.000,B 0.000,C 180.000,E1 0.000} C_DIS
LIN {X -32.628,Y 252.016,Z 140.000,A 0.000,B 0.000,C 180.000,E1 0.000} C_DIS
LIN {X -45.558,Y 250.002,Z 140.000,A 0.000,B 0.000,C 180.000,E1 0.000} C_DIS
LIN {X -58.368,Y 247.325,Z 140.000,A 0.000,B 0.000,C 180.000,E1 0.000} C_DIS
LIN {X -71.023,Y 243.993,Z 140.000,A 0.000,B 0.000,C 180.000,E1 0.000} C_DIS
LIN {X -83.489,Y 240.013,Z 140.000,A 0.000,B 0.000,C 180.000,E1 0.000} C_DIS
LIN {X -95.734,Y 235.396,Z 140.000,A 0.000,B 0.000,C 180.000,E1 0.000} C_DIS
LIN {X -107.725,Y 230.156,Z 140.000,A 0.000,B 0.000,C 180.000,E1 0.000} C_DIS
LIN {X -119.431,Y 224.306,Z 140.000,A 0.000,B 0.000,C 180.000,E1 0.000} C_DIS
LIN {X -130.819,Y 217.860,Z 140.000,A 0.000,B 0.000,C 180.000,E1 0.000} C_DIS
LIN {X -141.860,Y 210.838,Z 140.000,A 0.000,B 0.000,C 180.000,E1 0.000} C_DIS
LIN {X -152.526,Y 203.255,Z 140.000,A 0.000,B 0.000,C 180.000,E1 0.000} C_DIS
LIN {X -162.787,Y 195.134,Z 140.000,A 0.000,B 0.000,C 180.000,E1 0.000} C_DIS
LIN {X -172.617,Y 186.495,Z 140.000,A 0.000,B 0.000,C 180.000,E1 0.000} C_DIS
LIN {X -181.988,Y 177.361,Z 140.000,A 0.000,B 0.000,C 180.000,E1 0.000} C_DIS
LIN {X -190.878,Y 167.758,Z 140.000,A 0.000,B 0.000,C 180.000,E1 0.000} C_DIS
LIN {X -199.260,Y 157.709,Z 140.000,A 0.000,B 0.000,C 180.000,E1 0.000} C_DIS
LIN {X -207.114,Y 147.242,Z 140.000,A 0.000,B 0.000,C 180.000,E1 0.000} C_DIS
LIN {X -214.420,Y 136.385,Z 140.000,A 0.000,B 0.000,C 180.000,E1 0.000} C_DIS
LIN {X -221.157,Y 125.166,Z 140.000,A 0.000,B 0.000,C 180.000,E1 0.000} C_DIS
LIN {X -227.307,Y 113.614,Z 140.000,A 0.000,B 0.000,C 180.000,E1 0.000} C_DIS
LIN {X -232.855,Y 101.763,Z 140.000,A 0.000,B 0.000,C 180.000,E1 0.000} C_DIS
LIN {X -237.784,Y 89.641,Z 140.000,A 0.000,B 0.000,C 180.000,E1 0.000} C_DIS
LIN {X -242.083,Y 77.283,Z 140.000,A 0.000,B 0.000,C 180.000,E1 0.000} C_DIS
LIN {X -245.740,Y 64.716,Z 140.000,A 0.000,B 0.000,C 180.000,E1 0.000} C_DIS
LIN {X -248.746,Y 51.981,Z 140.000,A 0.000,B 0.000,C 180.000,E1 0.000} C_DIS
LIN {X -251.093,Y 39.106,Z 140.000,A 0.000,B 0.000,C 180.000,E1 0.000} C_DIS
LIN {X -252.773,Y 26.129,Z 140.000,A 0.000,B 0.000,C 180.000,E1 0.000} C_DIS
LIN {X -253.782,Y 13.082,Z 140.000,A 0.000,B 0.000,C 180.000,E1 0.000} C_DIS
LIN {X -254.119,Y 0.000,Z 140.000,A 0.000,B 0.000,C 180.000,E1 0.000} C_DIS
LIN {X -253.782,Y -13.082,Z 140.000,A 0.000,B 0.000,C 180.000,E1 0.000} C_DIS
LIN {X -252.773,Y -26.129,Z 140.000,A 0.000,B 0.000,C 180.000,E1 0.000} C_DIS
LIN {X -251.093,Y -39.106,Z 140.000,A 0.000,B 0.000,C 180.000,E1 0.000} C_DIS
LIN {X -248.746,Y -51.981,Z 140.000,A 0.000,B 0.000,C 180.000,E1 0.000} C_DIS
LIN {X -245.740,Y -64.716,Z 140.000,A 0.000,B 0.000,C 180.000,E1 0.000} C_DIS
LIN {X -242.083,Y -77.282,Z 140.000,A 0.000,B 0.000,C 180.000,E1 0.000} C_DIS
LIN {X -237.784,Y -89.641,Z 140.000,A 0.000,B 0.000,C 180.000,E1 0.000} C_DIS
LIN {X -232.855,Y -101.763,Z 140.000,A 0.000,B 0.000,C 180.000,E1 0.000} C_DIS
LIN {X -227.307,Y -113.614,Z 140.000,A 0.000,B 0.000,C 180.000,E1 0.000} C_DIS
LIN {X -221.157,Y -125.166,Z 140.000,A 0.000,B 0.000,C 180.000,E1 0.000} C_DIS
LIN {X -214.420,Y -136.385,Z 140.000,A 0.000,B 0.000,C 180.000,E1 0.000} C_DIS
LIN {X -207.114,Y -147.242,Z 140.000,A 0.000,B 0.000,C 180.000,E1 0.000} C_DIS
LIN {X -199.260,Y -157.709,Z 140.000,A 0.000,B 0.000,C 180.000,E1 0.000} C_DIS
LIN {X -190.878,Y -167.758,Z 140.000,A 0.000,B 0.000,C 180.000,E1 0.000} C_DIS
LIN {X -181.988,Y -177.361,Z 140.000,A 0.000,B 0.000,C 180.000,E1 0.000} C_DIS
LIN {X -172.616,Y -186.495,Z 140.000,A 0.000,B 0.000,C 180.000,E1 0.000} C_DIS
LIN {X -162.787,Y -195.133,Z 140.000,A 0.000,B 0.000,C 180.000,E1 0.000} C_DIS
LIN {X -152.526,Y -203.255,Z 140.000,A 0.000,B 0.000,C 180.000,E1 0.000} C_DIS
LIN {X -141.860,Y -210.838,Z 140.000,A 0.000,B 0.000,C 180.000,E1 0.000} C_DIS
LIN {X -130.819,Y -217.861,Z 140.000,A 0.000,B 0.000,C 180.000,E1 0.000} C_DIS
LIN {X -119.431,Y -224.306,Z 140.000,A 0.000,B 0.000,C 180.000,E1 0.000} C_DIS
LIN {X -107.725,Y -230.156,Z 140.000,A 0.000,B 0.000,C 180.000,E1 0.000} C_DIS
LIN {X -95.734,Y -235.396,Z 140.000,A 0.000,B 0.000,C 180.000,E1 0.000} C_DIS
LIN {X -83.489,Y -240.013,Z 140.000,A 0.000,B 0.000,C 180.000,E1 0.000} C_DIS
LIN {X -71.023,Y -243.993,Z 140.000,A 0.000,B 0.000,C 180.000,E1 0.000} C_DIS
LIN {X -58.368,Y -247.325,Z 140.000,A 0.000,B 0.000,C 180.000,E1 0.000} C_DIS
LIN {X -45.558,Y -250.002,Z 140.000,A 0.000,B 0.000,C 180.000,E1 0.000} C_DIS
LIN {X -32.628,Y -252.016,Z 140.000,A 0.000,B 0.000,C 180.000,E1 0.000} C_DIS
LIN {X -19.612,Y -253.361,Z 140.000,A 0.000,B 0.000,C 180.000,E1 0.000} C_DIS
LIN {X -6.543,Y -254.035,Z 140.000,A 0.000,B 0.000,C 180.000,E1 0.000} C_DIS
LIN {X 6.543,Y -254.035,Z 140.000,A 0.000,B 0.000,C 180.000,E1 0.000} C_DIS
LIN {X 19.612,Y -253.361,Z 140.000,A 0.000,B 0.000,C 180.000,E1 0.000} C_DIS
LIN {X 32.628,Y -252.016,Z 140.000,A 0.000,B 0.000,C 180.000,E1 0.000} C_DIS
LIN {X 45.558,Y -250.002,Z 140.000,A 0.000,B 0.000,C 180.000,E1 0.000} C_DIS
LIN {X 58.368,Y -247.325,Z 140.000,A 0.000,B 0.000,C 180.000,E1 0.000} C_DIS
LIN {X 71.023,Y -243.993,Z 140.000,A 0.000,B 0.000,C 180.000,E1 0.000} C_DIS
LIN {X 83.489,Y -240.013,Z 140.000,A 0.000,B 0.000,C 180.000,E1 0.000} C_DIS
LIN {X 95.734,Y -235.396,Z 140.000,A 0.000,B 0.000,C 180.000,E1 0.000} C_DIS
LIN {X 107.725,Y -230.156,Z 140.000,A 0.000,B 0.000,C 180.000,E1 0.000} C_DIS
LIN {X 119.431,Y -224.306,Z 140.000,A 0.000,B 0.000,C 180.000,E1 0.000} C_DIS
LIN {X 130.819,Y -217.860,Z 140.000,A 0.000,B 0.000,C 180.000,E1 0.000} C_DIS
LIN {X 141.860,Y -210.838,Z 140.000,A 0.000,B 0.000,C 180.000,E1 0.000} C_DIS
LIN {X 152.526,Y -203.255,Z 140.000,A 0.000,B 0.000,C 180.000,E1 0.000} C_DIS
LIN {X 162.787,Y -195.134,Z 140.000,A 0.000,B 0.000,C 180.000,E1 0.000} C_DIS
LIN {X 172.617,Y -186.495,Z 140.000,A 0.000,B 0.000,C 180.000,E1 0.000} C_DIS
LIN {X 181.988,Y -177.361,Z 140.000,A 0.000,B 0.000,C 180.000,E1 0.000} C_DIS
LIN {X 190.878,Y -167.758,Z 140.000,A 0.000,B 0.000,C 180.000,E1 0.000} C_DIS
LIN {X 199.260,Y -157.709,Z 140.000,A 0.000,B 0.000,C 180.000,E1 0.000} C_DIS
LIN {X 207.114,Y -147.242,Z 140.000,A 0.000,B 0.000,C 180.000,E1 0.000} C_DIS
LIN {X 214.420,Y -136.385,Z 140.000,A 0.000,B 0.000,C 180.000,E1 0.000} C_DIS
LIN {X 221.157,Y -125.166,Z 140.000,A 0.000,B 0.000,C 180.000,E1 0.000} C_DIS
LIN {X 227.307,Y -113.614,Z 140.000,A 0.000,B 0.000,C 180.000,E1 0.000} C_DIS
LIN {X 232.855,Y -101.763,Z 140.000,A 0.000,B 0.000,C 180.000,E1 0.000} C_DIS
LIN {X 237.784,Y -89.641,Z 140.000,A 0.000,B 0.000,C 180.000,E1 0.000} C_DIS
LIN {X 242.083,Y -77.283,Z 140.000,A 0.000,B 0.000,C 180.000,E1 0.000} C_DIS
LIN {X 245.740,Y -64.716,Z 140.000,A 0.000,B 0.000,C 180.000,E1 0.000} C_DIS
LIN {X 248.746,Y -51.981,Z 140.000,A 0.000,B 0.000,C 180.000,E1 0.000} C_DIS
LIN {X 251.093,Y -39.106,Z 140.000,A 0.000,B 0.000,C 180.000,E1 0.000} C_DIS
LIN {X 252.773,Y -26.129,Z 140.000,A 0.000,B 0.000,C 180.000,E1 0.000} C_DIS
LIN {X 253.782,Y -13.082,Z 140.000,A 0.000,B 0.000,C 180.000,E1 0.000} C_DIS
LIN {X 254.119,Y 0.000,Z 140.000,A 0.000,B 0.000,C 180.000,E1 0.000} C_DIS
LIN {X 253.782,Y 13.082,Z 140.000,A 0.000,B 0.000,C 180.000,E1 0.000} C_DIS
LIN {X 252.773,Y 26.129,Z 140.000,A 0.000,B 0.000,C 180.000,E1 0.000} C_DIS
;rapid-leaky
$VEL.CP=0.3
LIN {X 237.310,Y 24.531,Z 140.000,A 0.000,B 0.000,C 180.000,E1 0.000} C_DIS
;bead-perimeter_inner
$VEL.CP=0.65
LIN {X 235.733,Y 36.713,Z 140.000,A 0.000,B 0.000,C 180.000,E1 0.000} C_DIS
LIN {X 233.530,Y 48.800,Z 140.000,A 0.000,B 0.000,C 180.000,E1 0.000} C_DIS
LIN {X 230.708,Y 60.758,Z 140.000,A 0.000,B 0.000,C 180.000,E1 0.000} C_DIS
LIN {X 227.274,Y 72.555,Z 140.000,A 0.000,B 0.000,C 180.000,E1 0.000} C_DIS
LIN {X 223.238,Y 84.158,Z 140.000,A 0.000,B 0.000,C 180.000,E1 0.000} C_DIS
LIN {X 218.610,Y 95.538,Z 140.000,A 0.000,B 0.000,C 180.000,E1 0.000} C_DIS
LIN {X 213.402,Y 106.664,Z 140.000,A 0.000,B 0.000,C 180.000,E1 0.000} C_DIS
LIN {X 207.628,Y 117.509,Z 140.000,A 0.000,B 0.000,C 180.000,E1 0.000} C_DIS
LIN {X 201.304,Y 128.041,Z 140.000,A 0.000,B 0.000,C 180.000,E1 0.000} C_DIS
LIN {X 194.444,Y 138.235,Z 140.000,A 0.000,B 0.000,C 180.000,E1 0.000} C_DIS
LIN {X 187.071,Y 148.062,Z 140.000,A 0.000,B 0.000,C 180.000,E1 0.000} C_DIS
LIN {X 179.201,Y 157.495,Z 140.000,A 0.000,B 0.000,C 180.000,E1 0.000} C_DIS
LIN {X 170.855,Y 166.512,Z 140.000,A 0.000,B 0.000,C 180.000,E1 0.000} C_DIS
LIN {X 162.057,Y 175.087,Z 140.000,A 0.000,B 0.000,C 180.000,E1 0.000} C_DIS
LIN {X 152.830,Y 183.196,Z 140.000,A 0.000,B 0.000,C 180.000,E1 0.000} C_DIS
LIN {X 143.196,Y 190.821,Z 140.000,A 0.000,B 0.000,C 180.000,E1 0.000} C_DIS
LIN {X 133.182,Y 197.940,Z 140.000,A 0.000,B 0.000,C 180.000,E1 0.000} C_DIS
LIN {X 122.816,Y 204.534,Z 140.000,A 0.000,B 0.000,C 180.000,E1 0.000} C_DIS
LIN {X 112.125,Y 210.584,Z 140.000,A 0.000,B 0.000,C 180.000,E1 0.000} C_DIS
LIN {X 101.136,Y 216.077,Z 140.000,A 0.000,B 0.000,C 180.000,E1 0.000} C_DIS
LIN {X 89.878,Y 220.996,Z 140.000,A 0.000,B 0.000,C 180.000,E1 0.000} C_DIS
LIN {X 78.381,Y 225.331,Z 140.000,A 0.000,B 0.000,C 180.000,E1 0.000} C_DIS
LIN {X 66.678,Y 229.067,Z 140.000,A 0.000,B 0.000,C 180.000,E1 0.000} C_DIS
LIN {X 54.797,Y 232.196,Z 140.000,A 0.000,B 0.000,C 180.000,E1 0.000} C_DIS
LIN {X 42.771,Y 234.709,Z 140.000,A 0.000,B 0.000,C 180.000,E1 0.000} C_DIS
LIN {X 30.632,Y 236.600,Z 140.000,A 0.000,B 0.000,C 180.000,E1 0.000} C_DIS
LIN {X 18.413,Y 237.863,Z 140.000,A 0.000,B 0.000,C 180.000,E1 0.000} C_DIS
LIN {X 6.143,Y 238.495,Z 140.000,A 0.000,B 0.000,C 180.000,E1 0.000} C_DIS
LIN {X -6.143,Y 238.495,Z 140.000,A 0.000,B 0.000,C 180.000,E1 0.000} C_DIS
LIN {X -18.413,Y 237.863,Z 140.000,A 0.000,B 0.000,C 180.000,E1 0.000} C_DIS
LIN {X -30.632,Y 236.600,Z 140.000,A 0.000,B 0.000,C 180.000,E1 0.000} C_DIS
LIN {X -42.771,Y 234.709,Z 140.000,A 0.000,B 0.000,C 180.000,E1 0.000} C_DIS
LIN {X -54.797,Y 232.196,Z 140.000,A 0.000,B 0.000,C 180.000,E1 0.000} C_DIS
LIN {X -66.678,Y 229.067,Z 140.000,A 0.000,B 0.000,C 180.000,E1 0.000} C_DIS
LIN {X -78.381,Y 225.331,Z 140.000,A 0.000,B 0.000,C 180.000,E1 0.000} C_DIS
LIN {X -89.878,Y 220.996,Z 140.000,A 0.000,B 0.000,C 180.000,E1 0.000} C_DIS
LIN {X -101.136,Y 216.077,Z 140.000,A 0.000,B 0.000,C 180.000,E1 0.000} C_DIS
LIN {X -112.125,Y 210.584,Z 140.000,A 0.000,B 0.000,C 180.000,E1 0.000} C_DIS
LIN {X -122.817,Y 204.533,Z 140.000,A 0.000,B 0.000,C 180.000,E1 0.000} C_DIS
LIN {X -133.182,Y 197.941,Z 140.000,A 0.000,B 0.000,C 180.000,E1 0.000} C_DIS
LIN {X -143.196,Y 190.821,Z 140.000,A 0.000,B 0.000,C 180.000,E1 0.000} C_DIS
LIN {X -152.829,Y 183.197,Z 140.000,A 0.000,B 0.000,C 180.000,E1 0.000} C_DIS
LIN {X -162.057,Y 175.087,Z 140.000,A 0.000,B 0.000,C 180.000,E1 0.000} C_DIS
LIN {X -170.855,Y 166.512,Z 140.000,A 0.000,B 0.000,C 180.000,E1 0.000} C_DIS
LIN {X -179.201,Y 157.495,Z 140.000,A 0.000,B 0.000,C 180.000,E1 0.000} C_DIS
LIN {X -187.071,Y 148.062,Z 140.000,A 0.000,B 0.000,C 180.000,E1 0.000} C_DIS
LIN {X -194.444,Y 138.235,Z 140.000,A 0.000,B 0.000,C 180.000,E1 0.000} C_DIS
LIN {X -201.304,Y 128.041,Z 140.000,A 0.000,B 0.000,C 180.000,E1 0.000} C_DIS
LIN {X -207.628,Y 117.509,Z 140.000,A 0.000,B 0.000,C 180.000,E1 0.000} C_DIS
LIN {X -213.402,Y 106.664,Z 140.000,A 0.000,B 0.000,C 180.000,E1 0.000} C_DIS
LIN {X -218.610,Y 95.538,Z 140.000,A 0.000,B 0.000,C 180.000,E1 0.000} C_DIS
LIN {X -223.238,Y 84.158,Z 140.000,A 0.000,B 0.000,C 180.000,E1 0.000} C_DIS
LIN {X -227.274,Y 72.556,Z 140.000,A 0.000,B 0.000,C 180.000,E1 0.000} C_DIS
LIN {X -230.708,Y 60.758,Z 140.000,A 0.000,B 0.000,C 180.000,E1 0.000} C_DIS
LIN {X -233.530,Y 48.800,Z 140.000,A 0.000,B 0.000,C 180.000,E1 0.000} C_DIS
LIN {X -235.733,Y 36.713,Z 140.000,A 0.000,B 0.000,C 180.000,E1 0.000} C_DIS
LIN {X -237.310,Y 24.531,Z 140.000,A 0.000,B 0.000,C 180.000,E1 0.000} C_DIS
LIN {X -238.258,Y 12.282,Z 140.000,A 0.000,B 0.000,C 180.000,E1 0.000} C_DIS
LIN {X -238.574,Y 0.000,Z 140.000,A 0.000,B 0.000,C 180.000,E1 0.000} C_DIS
LIN {X -238.258,Y -12.282,Z 140.000,A 0.000,B 0.000,C 180.000,E1 0.000} C_DIS
LIN {X -237.310,Y -24.531,Z 140.000,A 0.000,B 0.000,C 180.000,E1 0.000} C_DIS
LIN {X -235.733,Y -36.713,Z 140.000,A 0.000,B 0.000,C 180.000,E1 0.000} C_DIS
LIN {X -233.530,Y -48.800,Z 140.000,A 0.000,B 0.000,C 180.000,E1 0.000} C_DIS
LIN {X -230.708,Y -60.758,Z 140.000,A 0.000,B 0.000,C 180.000,E1 0.000} C_DIS
LIN {X -227.274,Y -72.555,Z 140.000,A 0.000,B 0.000,C 180.000,E1 0.000} C_DIS
LIN {X -223.238,Y -84.158,Z 140.000,A 0.000,B 0.000,C 180.000,E1 0.000} C_DIS
LIN {X -218.610,Y -95.538,Z 140.000,A 0.000,B 0.000,C 180.000,E1 0.000} C_DIS
LIN {X -213.402,Y -106.664,Z 140.000,A 0.000,B 0.000,C 180.000,E1 0.000} C_DIS
LIN {X -207.628,Y -117.509,Z 140.000,A 0.000,B 0.000,C 180.000,E1 0.000} C_DIS
LIN {X -201.304,Y -128.041,Z 140.000,A 0.000,B 0.000,C 180.000,E1 0.000} C_DIS
LIN {X -194.444,Y -138.235,Z 140.000,A 0.000,B 0.000,C 180.000,E1 0.000} C_DIS
LIN {X -187.071,Y -148.062,Z 140.000,A 0.000,B 0.000,C 180.000,E1 0.000} C_DIS
LIN {X -179.201,Y -157.495,Z 140.000,A 0.000,B 0.000,C 180.000,E1 0.000} C_DIS
LIN {X -170.855,Y -166.512,Z 140.000,A 0.000,B 0.000,C 180.000,E1 0.000} C_DIS
LIN {X -162.057,Y -175.087,Z 140.000,A 0.000,B 0.000,C 180.000,E1 0.000} C_DIS
LIN {X -152.830,Y -183.196,Z 140.000,A 0.000,B 0.000,C 180.000,E1 0.000} C_DIS
LIN {X -143.196,Y -190.821,Z 140.000,A 0.000,B 0.000,C 180.000,E1 0.000} C_DIS
LIN {X -133.182,Y -197.940,Z 140.000,A 0.000,B 0.000,C 180.000,E1 0.000} C_DIS
LIN {X -122.816,Y -204.534,Z 140.000,A 0.000,B 0.000,C 180.000,E1 0.000} C_DIS
LIN {X -112.125,Y -210.584,Z 140.000,A 0.000,B 0.000,C 180.000,E1 0.000} C_DIS
LIN {X -101.136,Y -216.077,Z 140.000,A 0.000,B 0.000,C 180.000,E1 0.000} C_DIS
LIN {X -89.878,Y -220.996,Z 140.000,A 0.000,B 0.000,C 180.000,E1 0.000} C_DIS
LIN {X -78.381,Y -225.331,Z 140.000,A 0.000,B 0.000,C 180.000,E1 0.000} C_DIS
LIN {X -66.678,Y -229.067,Z 140.000,A 0.000,B 0.000,C 180.000,E1 0.000} C_DIS
LIN {X -54.797,Y -232.196,Z 140.000,A 0.000,B 0.000,C 180.000,E1 0.000} C_DIS
LIN {X -42.771,Y -234.709,Z 140.000,A 0.000,B 0.000,C 180.000,E1 0.000} C_DIS
LIN {X -30.632,Y -236.600,Z 140.000,A 0.000,B 0.000,C 180.000,E1 0.000} C_DIS
LIN {X -18.413,Y -237.863,Z 140.000,A 0.000,B 0.000,C 180.000,E1 0.000} C_DIS
LIN {X -6.143,Y -238.495,Z 140.000,A 0.000,B 0.000,C 180.000,E1 0.000} C_DIS
LIN {X 6.143,Y -238.495,Z 140.000,A 0.000,B 0.000,C 180.000,E1 0.000} C_DIS
LIN {X 18.413,Y -237.863,Z 140.000,A 0.000,B 0.000,C 180.000,E1 0.000} C_DIS
LIN {X 30.632,Y -236.600,Z 140.000,A 0.000,B 0.000,C 180.000,E1 0.000} C_DIS
LIN {X 42.771,Y -234.709,Z 140.000,A 0.000,B 0.000,C 180.000,E1 0.000} C_DIS
LIN {X 54.797,Y -232.196,Z 140.000,A 0.000,B 0.000,C 180.000,E1 0.000} C_DIS
LIN {X 66.678,Y -229.067,Z 140.000,A 0.000,B 0.000,C 180.000,E1 0.000} C_DIS
LIN {X 78.381,Y -225.331,Z 140.000,A 0.000,B 0.000,C 180.000,E1 0.000} C_DIS
LIN {X 89.878,Y -220.996,Z 140.000,A 0.000,B 0.000,C 180.000,E1 0.000} C_DIS
LIN {X 101.136,Y -216.077,Z 140.000,A 0.000,B 0.000,C 180.000,E1 0.000} C_DIS
LIN {X 112.125,Y -210.584,Z 140.000,A 0.000,B 0.000,C 180.000,E1 0.000} C_DIS
LIN {X 122.817,Y -204.533,Z 140.000,A 0.000,B 0.000,C 180.000,E1 0.000} C_DIS
LIN {X 133.182,Y -197.941,Z 140.000,A 0.000,B 0.000,C 180.000,E1 0.000} C_DIS
LIN {X 143.196,Y -190.821,Z 140.000,A 0.000,B 0.000,C 180.000,E1 0.000} C_DIS
LIN {X 152.829,Y -183.197,Z 140.000,A 0.000,B 0.000,C 180.000,E1 0.000} C_DIS
LIN {X 162.057,Y -175.087,Z 140.000,A 0.000,B 0.000,C 180.000,E1 0.000} C_DIS
LIN {X 170.855,Y -166.512,Z 140.000,A 0.000,B 0.000,C 180.000,E1 0.000} C_DIS
LIN {X 179.201,Y -157.495,Z 140.000,A 0.000,B 0.000,C 180.000,E1 0.000} C_DIS
LIN {X 187.071,Y -148.062,Z 140.000,A 0.000,B 0.000,C 180.000,E1 0.000} C_DIS
LIN {X 194.444,Y -138.235,Z 140.000,A 0.000,B 0.000,C 180.000,E1 0.000} C_DIS
LIN {X 201.304,Y -128.041,Z 140.000,A 0.000,B 0.000,C 180.000,E1 0.000} C_DIS
LIN {X 207.628,Y -117.509,Z 140.000,A 0.000,B 0.000,C 180.000,E1 0.000} C_DIS
LIN {X 213.402,Y -106.664,Z 140.000,A 0.000,B 0.000,C 180.000,E1 0.000} C_DIS
LIN {X 218.610,Y -95.538,Z 140.000,A 0.000,B 0.000,C 180.000,E1 0.000} C_DIS
LIN {X 223.238,Y -84.158,Z 140.000,A 0.000,B 0.000,C 180.000,E1 0.000} C_DIS
LIN {X 227.274,Y -72.556,Z 140.000,A 0.000,B 0.000,C 180.000,E1 0.000} C_DIS
LIN {X 230.708,Y -60.758,Z 140.000,A 0.000,B 0.000,C 180.000,E1 0.000} C_DIS
LIN {X 233.530,Y -48.800,Z 140.000,A 0.000,B 0.000,C 180.000,E1 0.000} C_DIS
LIN {X 235.733,Y -36.713,Z 140.000,A 0.000,B 0.000,C 180.000,E1 0.000} C_DIS
LIN {X 237.310,Y -24.531,Z 140.000,A 0.000,B 0.000,C 180.000,E1 0.000} C_DIS
LIN {X 238.258,Y -12.282,Z 140.000,A 0.000,B 0.000,C 180.000,E1 0.000} C_DIS
LIN {X 238.574,Y 0.000,Z 140.000,A 0.000,B 0.000,C 180.000,E1 0.000} C_DIS
LIN {X 238.258,Y 12.282,Z 140.000,A 0.000,B 0.000,C 180.000,E1 0.000} C_DIS
LIN {X 237.310,Y 24.531,Z 140.000,A 0.000,B 0.000,C 180.000,E1 0.000} C_DIS
;rapid-leaky
$VEL.CP=0.3
LIN {X 207.668,Y -74.861,Z 140.000,A 0.000,B 0.000,C 180.000,E1 0.000} C_DIS
;bead-sparse_infill
$VEL.CP=0.65
LIN {X 74.847,Y -207.683,Z 140.000,A 0.000,B 0.000,C 180.000,E1 0.000} C_DIS
LIN {X 72.544,Y -208.551,Z 140.000,A 0.000,B 0.000,C 180.000,E1 0.000} C_DIS
LIN {X 61.713,Y -212.009,Z 140.000,A 0.000,B 0.000,C 180.000,E1 0.000} C_DIS
LIN {X 50.717,Y -214.905,Z 140.000,A 0.000,B 0.000,C 180.000,E1 0.000} C_DIS
LIN {X 39.586,Y -217.231,Z 140.000,A 0.000,B 0.000,C 180.000,E1 0.000} C_DIS
LIN {X 28.351,Y -218.981,Z 140.000,A 0.000,B 0.000,C 180.000,E1 0.000} C_DIS
LIN {X 17.042,Y -220.150,Z 140.000,A 0.000,B 0.000,C 180.000,E1 0.000} C_DIS
LIN {X 5.686,Y -220.735,Z 140.000,A 0.000,B 0.000,C 180.000,E1 0.000} C_DIS
LIN {X -5.686,Y -220.735,Z 140.000,A 0.000,B 0.000,C 180.000,E1 0.000} C_DIS
LIN {X -17.042,Y -220.150,Z 140.000,A 0.000,B 0.000,C 180.000,E1 0.000} C_DIS
LIN {X -28.351,Y -218.981,Z 140.000,A 0.000,B 0.000,C 180.000,E1 0.000} C_DIS
LIN {X -39.586,Y -217.231,Z 140.000,A 0.000,B 0.000,C 180.000,E1 0.000} C_DIS
LIN {X -50.717,Y -214.905,Z 140.000,A 0.000,B 0.000,C 180.000,E1 0.000} C_DIS
LIN {X -61.713,Y -212.009,Z 140.000,A 0.000,B 0.000,C 180.000,E1 0.000} C_DIS
LIN {X -72.544,Y -208.551,Z 140.000,A 0.000,B 0.000,C 180.000,E1 0.000} C_DIS
LIN {X -80.137,Y -205.689,Z 140.000,A 0.000,B 0.000,C 180.000,E1 0.000} C_DIS
LIN {X 205.697,Y 80.146,Z 140.000,A 0.000,B 0.000,C 180.000,E1 0.000} C_DIS
LIN {X 202.331,Y 88.424,Z 140.000,A 0.000,B 0.000,C 180.000,E1 0.000} C_DIS
LIN {X 197.511,Y 98.721,Z 140.000,A 0.000,B 0.000,C 180.000,E1 0.000} C_DIS
LIN {X 192.166,Y 108.759,Z 140.000,A 0.000,B 0.000,C 180.000,E1 0.000} C_DIS
LIN {X 186.313,Y 118.506,Z 140.000,A 0.000,B 0.000,C 180.000,E1 0.000} C_DIS
LIN {X 179.965,Y 127.941,Z 140.000,A 0.000,B 0.000,C 180.000,E1 0.000} C_DIS
LIN {X 173.140,Y 137.037,Z 140.000,A 0.000,B 0.000,C 180.000,E1 0.000} C_DIS
LIN {X 165.857,Y 145.767,Z 140.000,A 0.000,B 0.000,C 180.000,E1 0.000} C_DIS
LIN {X 158.132,Y 154.112,Z 140.000,A 0.000,B 0.000,C 180.000,E1 0.000} C_DIS
LIN {X 149.989,Y 162.049,Z 140.000,A 0.000,B 0.000,C 180.000,E1 0.000} C_DIS
LIN {X 141.449,Y 169.554,Z 140.000,A 0.000,B 0.000,C 180.000,E1 0.000} C_DIS
LIN {X 139.595,Y 171.021,Z 140.000,A 0.000,B 0.000,C 180.000,E1 0.000} C_DIS
LIN {X -171.013,Y -139.587,Z 140.000,A 0.000,B 0.000,C 180.000,E1 0.000} C_DIS
LIN {X -173.140,Y -137.037,Z 140.000,A 0.000,B 0.000,C 180.000,E1 0.000} C_DIS
LIN {X -179.965,Y -127.941,Z 140.000,A 0.000,B 0.000,C 180.000,E1 0.000} C_DIS
LIN {X -186.313,Y -118.506,Z 140.000,A 0.000,B 0.000,C 180.000,E1 0.000} C_DIS
LIN {X -192.166,Y -108.759,Z 140.000,A 0.000,B 0.000,C 180.000,E1 0.000} C_DIS
LIN {X -197.511,Y -98.721,Z 140.000,A 0.000,B 0.000,C 180.000,E1 0.000} C_DIS
LIN {X -202.331,Y -88.424,Z 140.000,A 0.000,B 0.000,C 180.000,E1 0.000} C_DIS
LIN {X -206.614,Y -77.891,Z 140.000,A 0.000,B 0.000,C 180.000,E1 0.000} C_DIS
LIN {X -210.350,Y -67.153,Z 140.000,A 0.000,B 0.000,C 180.000,E1 0.000} C_DIS
LIN {X -213.528,Y -56.234,Z 140.000,A 0.000,B 0.000,C 180.000,E1 0.000} C_DIS
LIN {X -216.140,Y -45.166,Z 140.000,A 0.000,B 0.000,C 180.000,E1 0.000} C_DIS
LIN {X -218.179,Y -33.979,Z 140.000,A 0.000,B 0.000,C 180.000,E1 0.000} C_DIS
LIN {X -218.661,Y -30.257,Z 140.000,A 0.000,B 0.000,C 180.000,E1 0.000} C_DIS
LIN {X 30.277,Y 218.681,Z 140.000,A 0.000,B 0.000,C 180.000,E1 0.000} C_DIS
;rapid-leaky
$VEL.CP=0.3
LIN {X 138.786,Y 206.266,Z 150.000,A 0.000,B 0.000,C 180.000,E1 0.000} C_DIS
;bead-perimeter_outer
$VEL.CP=0.63
LIN {X 127.983,Y 213.138,Z 150.000,A 0.000,B 0.000,C 180.000,E1 0.000} C_DIS
LIN {X 116.842,Y 219.443,Z 150.000,A 0.000,B 0.000,C 180.000,E1 0.000} C_DIS
LIN {X 105.389,Y 225.167,Z 150.000,A 0.000,B 0.000,C 180.000,E1 0.000} C_DIS
LIN {X 93.658,Y 230.293,Z 150.000,A 0.000,B 0.000,C 180.000,E1 0.000} C_DIS
LIN {X 81.679,Y 234.810,Z 150.000,A 0.000,B 0.000,C 180.000,E1 0.000} C_DIS
LIN {X 69.482,Y 238.703,Z 150.000,A 0.000,B 0.000,C 180.000,E1 0.000} C_DIS
LIN {X 57.102,Y 241.964,Z 150.000,A 0.000,B 0.000,C 180.000,E1 0.000} C_DIS
LIN {X 44.571,Y 244.582,Z 150.000,A 0.000,B 0.000,C 180.000,E1 0.000} C_DIS
LIN {X 31.920,Y 246.553,Z 150.000,A 0.000,B 0.000,C 180.000,E1 0.000} C_DIS
LIN {X 19.186,Y 247.869,Z 150.000,A 0.000,B 0.000,C 180.000,E1 0.000} C_DIS
LIN {X 6.401,Y 248.528,Z 150.000,A 0.000,B 0.000,C 180.000,E1 0.000} C_DIS
LIN {X -6.401,Y 248.528,Z 150.000,A 0.000,B 0.000,C 180.000,E1 0.000} C_DIS
LIN {X -19.186,Y 247.869,Z 150.000,A 0.000,B 0.000,C 180.000,E1 0.000} C_DIS
LIN {X -31.920,Y 246.553,Z 150.000,A 0.000,B 0.000,C 180.000,E1 0.000} C_DIS
LIN {X -44.571,Y 244.582,Z 150.000,A 0.000,B 0.000,C 180.000,E1 0.000} C_DIS
LIN {X -57.102,Y 241.964,Z 150.000,A 0.000,B 0.000,C 180.000,E1 0.000} C_DIS
LIN {X -69.482,Y 238.703,Z 150.000,A 0.000,B 0.000,C 180.000,E1 0.000} C_DIS
LIN {X -81.679,Y 234.810,Z 150.000,A 0.000,B 0.000,C 180.000,E1 0.000} C_DIS
LIN {X -93.658,Y 230.293,Z 150.000,A 0.000,B 0.000,C 180.000,E1 0.000} C_DIS
LIN {X -105.389,Y 225.167,Z 150.000,A 0.000,B 0.000,C 180.000,E1 0.000} C_DIS
LIN {X -116.842,Y 219.443,Z 150.000,A 0.000,B 0.000,C 180.000,E1 0.000} C_DIS
LIN {X -127.983,Y 213.138,Z 150.000,A 0.000,B 0.000,C 180.000,E1 0.000} C_DIS
LIN {X -138.786,Y 206.266,Z 150.000,A 0.000,B 0.000,C 180.000,E1 0.000} C_DIS
LIN {X -149.220,Y 198.849,Z 150.000,A 0.000,B 0.000,C 180.000,E1 0.000} C_DIS
LIN {X -159.258,Y 190.903,Z 150.000,A 0.000,B 0.000,C 180.000,E1 0.000} C_DIS
LIN {X -168.875,Y 182.451,Z 150.000,A 0.000,B 0.000,C 180.000,E1 0.000} C_DIS
LIN {X -178.043,Y 173.516,Z 150.000,A 0.000,B 0.000,C 180.000,E1 0.000} C_DIS
LIN {X -186.740,Y 164.121,Z 150.000,A 0.000,B 0.000,C 180.000,E1 0.000} C_DIS
LIN {X -194.940,Y 154.290,Z 150.000,A 0.000,B 0.000,C 180.000,E1 0.000} C_DIS
LIN {X -202.624,Y 144.050,Z 150.000,A 0.000,B 0.000,C 180.000,E1 0.000} C_DIS
LIN {X -209.772,Y 133.429,Z 150.000,A 0.000,B 0.000,C 180.000,E1 0.000} C_DIS
LIN {X -216.361,Y 122.452,Z 150.000,A 0.000,B 0.000,C 180.000,E1 0.000} C_DIS
LIN {X -222.379,Y 111.151,Z 150.000,A 0.000,B 0.000,C 180.000,E1 0.000} C_DIS
LIN {X -227.807,Y 99.557,Z 150.000,A 0.000,B 0.000,C 180.000,E1 0.000} C_DIS
LIN {X -232.629,Y 87.697,Z 150.000,A 0.000,B 0.000,C 180.000,E1 0.000} C_DIS
LIN {X -233.983,Y 83.808,Z 150.000,A 0.000,B 0.000,C 180.000,E1 0.000} C_DIS
LIN {X -236.835,Y 75.606,Z 150.000,A 0.000,B 0.000,C 180.000,E1 0.000} C_DIS
LIN {X -240.413,Y 63.314,Z 150.000,A 0.000,B 0.000,C 180.000,E1 0.000} C_DIS
LIN {X -243.354,Y 50.854,Z 150.000,A 0.000,B 0.000,C 180.000,E1 0.000} C_DIS
LIN {X -245.649,Y 38.259,Z 150.000,A 0.000,B 0.000,C 180.000,E1 0.000} C_DIS
LIN {X -247.293,Y 25.562,Z 150.000,A 0.000,B 0.000,C 180.000,E1 0.000} C_DIS
LIN {X -248.281,Y 12.799,Z 150.000,A 0.000,B 0.000,C 180.000,E1 0.000} C_DIS
LIN {X -248.610,Y 0.000,Z 150.000,A 0.000,B 0.000,C 180.000,E1 0.000} C_DIS
LIN {X -248.281,Y -12.799,Z 150.000,A 0.000,B 0.000,C 180.000,E1 0.000} C_DIS
LIN {X -247.293,Y -25.563,Z 150.000,A 0.000,B 0.000,C 180.000,E1 0.000} C_DIS
LIN {X -246.765,Y -29.644,Z 150.000,A 0.000,B 0.000,C 180.000,E1 0.000} C_DIS
LIN {X -245.649,Y -38.259,Z 150.000,A 0.000,B 0.000,C 180.000,E1 0.000} C_DIS
LIN {X -243.354,Y -50.854,Z 150.000,A 0.000,B 0.000,C 180.000,E1 0.000} C_DIS
LIN {X -240.413,Y -63.314,Z 150.000,A 0.000,B 0.000,C 180.000,E1 0.000} C_DIS
LIN {X -236.835,Y -75.606,Z 150.000,A 0.000,B 0.000,C 180.000,E1 0.000} C_DIS
LIN {X -232.629,Y -87.697,Z 150.000,A 0.000,B 0.000,C 180.000,E1 0.000} C_DIS
LIN {X -227.807,Y -99.557,Z 150.000,A 0.000,B 0.000,C 180.000,E1 0.000} C_DIS
LIN {X -222.379,Y -111.151,Z 150.000,A 0.000,B 0.000,C 180.000,E1 0.000} C_DIS
LIN {X -216.361,Y -122.452,Z 150.000,A 0.000,B 0.000,C 180.000,E1 0.000} C_DIS
LIN {X -209.772,Y -133.429,Z 150.000,A 0.000,B 0.000,C 180.000,E1 0.000} C_DIS
LIN {X -202.624,Y -144.050,Z 150.000,A 0.000,B 0.000,C 180.000,E1 0.000} C_DIS
LIN {X -194.940,Y -154.290,Z 150.000,A 0.000,B 0.000,C 180.000,E1 0.000} C_DIS
LIN {X -186.740,Y -164.121,Z 150.000,A 0.000,B 0.000,C 180.000,E1 0.000} C_DIS
LIN {X -178.043,Y -173.516,Z 150.000,A 0.000,B 0.000,C 180.000,E1 0.000} C_DIS
LIN {X -168.875,Y -182.451,Z 150.000,A 0.000,B 0.000,C 180.000,E1 0.000} C_DIS
LIN {X -159.258,Y -190.903,Z 150.000,A 0.000,B 0.000,C 180.000,E1 0.000} C_DIS
LIN {X -149.220,Y -198.849,Z 150.000,A 0.000,B 0.000,C 180.000,E1 0.000} C_DIS
LIN {X -138.786,Y -206.266,Z 150.000,A 0.000,B 0.000,C 180.000,E1 0.000} C_DIS
LIN {X -127.983,Y -213.138,Z 150.000,A 0.000,B 0.000,C 180.000,E1 0.000} C_DIS
LIN {X -116.842,Y -219.443,Z 150.000,A 0.000,B 0.000,C 180.000,E1 0.000} C_DIS
LIN {X -105.389,Y -225.167,Z 150.000,A 0.000,B 0.000,C 180.000,E1 0.000} C_DIS
LIN {X -93.658,Y -230.293,Z 150.000,A 0.000,B 0.000,C 180.000,E1 0.000} C_DIS
LIN {X -81.679,Y -234.810,Z 150.000,A 0.000,B 0.000,C 180.000,E1 0.000} C_DIS
LIN {X -69.482,Y -238.703,Z 150.000,A 0.000,B 0.000,C 180.000,E1 0.000} C_DIS
LIN {X -57.102,Y -241.964,Z 150.000,A 0.000,B 0.000,C 180.000,E1 0.000} C_DIS
LIN {X -44.571,Y -244.582,Z 150.000,A 0.000,B 0.000,C 180.000,E1 0.000} C_DIS
LIN {X -31.920,Y -246.553,Z 150.000,A 0.000,B 0.000,C 180.000,E1 0.000} C_DIS
LIN {X -19.186,Y -247.869,Z 150.000,A 0.000,B 0.000,C 180.000,E1 0.000} C_DIS
LIN {X -6.401,Y -248.528,Z 150.000,A 0.000,B 0.000,C 180.000,E1 0.000} C_DIS
LIN {X 6.401,Y -248.528,Z 150.000,A 0.000,B 0.000,C 180.000,E1 0.000} C_DIS
LIN {X 19.186,Y -247.869,Z 150.000,A 0.000,B 0.000,C 180.000,E1 0.000} C_DIS
LIN {X 31.920,Y -246.553,Z 150.000,A 0.000,B 0.000,C 180.000,E1 0.000} C_DIS
LIN {X 44.571,Y -244.582,Z 150.000,A 0.000,B 0.000,C 180.000,E1 0.000} C_DIS
LIN {X 57.102,Y -241.964,Z 150.000,A 0.000,B 0.000,C 180.000,E1 0.000} C_DIS
LIN {X 69.482,Y -238.703,Z 150.000,A 0.000,B 0.000,C 180.000,E1 0.000} C_DIS
LIN {X 81.679,Y -234.810,Z 150.000,A 0.000,B 0.000,C 180.000,E1 0.000} C_DIS
LIN {X 93.658,Y -230.293,Z 150.000,A 0.000,B 0.000,C 180.000,E1 0.000} C_DIS
LIN {X 105.389,Y -225.167,Z 150.000,A 0.000,B 0.000,C 180.000,E1 0.000} C_DIS
LIN {X 116.842,Y -219.443,Z 150.000,A 0.000,B 0.000,C 180.000,E1 0.000} C_DIS
LIN {X 127.983,Y -213.138,Z 150.000,A 0.000,B 0.000,C 180.000,E1 0.000} C_DIS
LIN {X 138.786,Y -206.266,Z 150.000,A 0.000,B 0.000,C 180.000,E1 0.000} C_DIS
LIN {X 149.220,Y -198.849,Z 150.000,A 0.000,B 0.000,C 180.000,E1 0.000} C_DIS
LIN {X 159.258,Y -190.903,Z 150.000,A 0.000,B 0.000,C 180.000,E1 0.000} C_DIS
LIN {X 168.875,Y -182.451,Z 150.000,A 0.000,B 0.000,C 180.000,E1 0.000} C_DIS
LIN {X 178.043,Y -173.516,Z 150.000,A 0.000,B 0.000,C 180.000,E1 0.000} C_DIS
LIN {X 186.740,Y -164.121,Z 150.000,A 0.000,B 0.000,C 180.000,E1 0.000} C_DIS
LIN {X 194.940,Y -154.290,Z 150.000,A 0.000,B 0.000,C 180.000,E1 0.000} C_DIS
LIN {X 202.624,Y -144.050,Z 150.000,A 0.000,B 0.000,C 180.000,E1 0.000} C_DIS
LIN {X 209.772,Y -133.429,Z 150.000,A 0.000,B 0.000,C 180.000,E1 0.000} C_DIS
LIN {X 216.361,Y -122.452,Z 150.000,A 0.000,B 0.000,C 180.000,E1 0.000} C_DIS
LIN {X 222.379,Y -111.151,Z 150.000,A 0.000,B 0.000,C 180.000,E1 0.000} C_DIS
LIN {X 227.807,Y -99.557,Z 150.000,A 0.000,B 0.000,C 180.000,E1 0.000} C_DIS
LIN {X 232.629,Y -87.697,Z 150.000,A 0.000,B 0.000,C 180.000,E1 0.000} C_DIS
LIN {X 236.835,Y -75.606,Z 150.000,A 0.000,B 0.000,C 180.000,E1 0.000} C_DIS
LIN {X 240.413,Y -63.314,Z 150.000,A 0.000,B 0.000,C 180.000,E1 0.000} C_DIS
LIN {X 243.354,Y -50.854,Z 150.000,A 0.000,B 0.000,C 180.000,E1 0.000} C_DIS
LIN {X 245.649,Y -38.259,Z 150.000,A 0.000,B 0.000,C 180.000,E1 0.000} C_DIS
LIN {X 247.293,Y -25.562,Z 150.000,A 0.000,B 0.000,C 180.000,E1 0.000} C_DIS
LIN {X 248.281,Y -12.799,Z 150.000,A 0.000,B 0.000,C 180.000,E1 0.000} C_DIS
LIN {X 248.610,Y 0.000,Z 150.000,A 0.000,B 0.000,C 180.000,E1 0.000} C_DIS
LIN {X 248.281,Y 12.799,Z 150.000,A 0.000,B 0.000,C 180.000,E1 0.000} C_DIS
LIN {X 247.293,Y 25.563,Z 150.000,A 0.000,B 0.000,C 180.000,E1 0.000} C_DIS
LIN {X 245.649,Y 38.259,Z 150.000,A 0.000,B 0.000,C 180.000,E1 0.000} C_DIS
LIN {X 243.354,Y 50.854,Z 150.000,A 0.000,B 0.000,C 180.000,E1 0.000} C_DIS
LIN {X 240.413,Y 63.314,Z 150.000,A 0.000,B 0.000,C 180.000,E1 0.000} C_DIS
LIN {X 236.835,Y 75.606,Z 150.000,A 0.000,B 0.000,C 180.000,E1 0.000} C_DIS
LIN {X 232.629,Y 87.697,Z 150.000,A 0.000,B 0.000,C 180.000,E1 0.000} C_DIS
LIN {X 227.807,Y 99.557,Z 150.000,A 0.000,B 0.000,C 180.000,E1 0.000} C_DIS
LIN {X 222.379,Y 111.151,Z 150.000,A 0.000,B 0.000,C 180.000,E1 0.000} C_DIS
LIN {X 216.361,Y 122.452,Z 150.000,A 0.000,B 0.000,C 180.000,E1 0.000} C_DIS
LIN {X 209.772,Y 133.429,Z 150.000,A 0.000,B 0.000,C 180.000,E1 0.000} C_DIS
LIN {X 202.624,Y 144.050,Z 150.000,A 0.000,B 0.000,C 180.000,E1 0.000} C_DIS
LIN {X 194.940,Y 154.290,Z 150.000,A 0.000,B 0.000,C 180.000,E1 0.000} C_DIS
LIN {X 186.740,Y 164.121,Z 150.000,A 0.000,B 0.000,C 180.000,E1 0.000} C_DIS
LIN {X 178.043,Y 173.516,Z 150.000,A 0.000,B 0.000,C 180.000,E1 0.000} C_DIS
LIN {X 168.875,Y 182.451,Z 150.000,A 0.000,B 0.000,C 180.000,E1 0.000} C_DIS
LIN {X 159.258,Y 190.903,Z 150.000,A 0.000,B 0.000,C 180.000,E1 0.000} C_DIS
LIN {X 149.220,Y 198.849,Z 150.000,A 0.000,B 0.000,C 180.000,E1 0.000} C_DIS
LIN {X 138.786,Y 206.266,Z 150.000,A 0.000,B 0.000,C 180.000,E1 0.000} C_DIS
;rapid-leaky
$VEL.CP=0.3
LIN {X 130.108,Y 193.369,Z 150.000,A 0.000,B 0.000,C 180.000,E1 0.000} C_DIS
;bead-perimeter_inner
$VEL.CP=0.63
LIN {X 119.981,Y 199.810,Z 150.000,A 0.000,B 0.000,C 180.000,E1 0.000} C_DIS
LIN {X 109.536,Y 205.722,Z 150.000,A 0.000,B 0.000,C 180.000,E1 0.000} C_DIS
LIN {X 98.800,Y 211.088,Z 150.000,A 0.000,B 0.000,C 180.000,E1 0.000} C_DIS
LIN {X 87.802,Y 215.893,Z 150.000,A 0.000,B 0.000,C 180.000,E1 0.000} C_DIS
LIN {X 76.572,Y 220.127,Z 150.000,A 0.000,B 0.000,C 180.000,E1 0.000} C_DIS
LIN {X 65.137,Y 223.777,Z 150.000,A 0.000,B 0.000,C 180.000,E1 0.000} C_DIS
LIN {X 53.532,Y 226.835,Z 150.000,A 0.000,B 0.000,C 180.000,E1 0.000} C_DIS
LIN {X 41.784,Y 229.289,Z 150.000,A 0.000,B 0.000,C 180.000,E1 0.000} C_DIS
LIN {X 29.924,Y 231.137,Z 150.000,A 0.000,B 0.000,C 180.000,E1 0.000} C_DIS
LIN {X 17.987,Y 232.371,Z 150.000,A 0.000,B 0.000,C 180.000,E1 0.000} C_DIS
LIN {X 6.001,Y 232.988,Z 150.000,A 0.000,B 0.000,C 180.000,E1 0.000} C_DIS
LIN {X -6.001,Y 232.988,Z 150.000,A 0.000,B 0.000,C 180.000,E1 0.000} C_DIS
LIN {X -17.987,Y 232.371,Z 150.000,A 0.000,B 0.000,C 180.000,E1 0.000} C_DIS
LIN {X -29.924,Y 231.137,Z 150.000,A 0.000,B 0.000,C 180.000,E1 0.000} C_DIS
LIN {X -41.784,Y 229.289,Z 150.000,A 0.000,B 0.000,C 180.000,E1 0.000} C_DIS
LIN {X -53.532,Y 226.835,Z 150.000,A 0.000,B 0.000,C 180.000,E1 0.000} C_DIS
LIN {X -65.137,Y 223.777,Z 150.000,A 0.000,B 0.000,C 180.000,E1 0.000} C_DIS
LIN {X -76.572,Y 220.127,Z 150.000,A 0.000,B 0.000,C 180.000,E1 0.000} C_DIS
LIN {X -87.802,Y 215.893,Z 150.000,A 0.000,B 0.000,C 180.000,E1 0.000} C_DIS
LIN {X -98.800,Y 211.088,Z 150.000,A 0.000,B 0.000,C 180.000,E1 0.000} C_DIS
LIN {X -109.536,Y 205.722,Z 150.000,A 0.000,B 0.000,C 180.000,E1 0.000} C_DIS
LIN {X -119.981,Y 199.810,Z 150.000,A 0.000,B 0.000,C 180.000,E1 0.000} C_DIS
LIN {X -130.108,Y 193.369,Z 150.000,A 0.000,B 0.000,C 180.000,E1 0.000} C_DIS
LIN {X -139.889,Y 186.416,Z 150.000,A 0.000,B 0.000,C 180.000,E1 0.000} C_DIS
LIN {X -149.299,Y 178.967,Z 150.000,A 0.000,B 0.000,C 180.000,E1 0.000} C_DIS
LIN {X -158.316,Y 171.043,Z 150.000,A 0.000,B 0.000,C 180.000,E1 0.000} C_DIS
LIN {X -166.911,Y 162.666,Z 150.000,A 0.000,B 0.000,C 180.000,E1 0.000} C_DIS
LIN {X -175.063,Y 153.859,Z 150.000,A 0.000,B 0.000,C 180.000,E1 0.000} C_DIS
LIN {X -182.751,Y 144.643,Z 150.000,A 0.000,B 0.000,C 180.000,E1 0.000} C_DIS
LIN {X -189.955,Y 135.043,Z 150.000,A 0.000,B 0.000,C 180.000,E1 0.000} C_DIS
LIN {X -196.655,Y 125.086,Z 150.000,A 0.000,B 0.000,C 180.000,E1 0.000} C_DIS
LIN {X -202.832,Y 114.796,Z 150.000,A 0.000,B 0.000,C 180.000,E1 0.000} C_DIS
LIN {X -208.475,Y 104.200,Z 150.000,A 0.000,B 0.000,C 180.000,E1 0.000} C_DIS
LIN {X -213.562,Y 93.332,Z 150.000,A 0.000,B 0.000,C 180.000,E1 0.000} C_DIS
LIN {X -218.084,Y 82.213,Z 150.000,A 0.000,B 0.000,C 180.000,E1 0.000} C_DIS
LIN {X -219.306,Y 78.700,Z 150.000,A 0.000,B 0.000,C 180.000,E1 0.000} C_DIS
LIN {X -222.026,Y 70.879,Z 150.000,A 0.000,B 0.000,C 180.000,E1 0.000} C_DIS
LIN {X -225.381,Y 59.355,Z 150.000,A 0.000,B 0.000,C 180.000,E1 0.000} C_DIS
LIN {X -228.138,Y 47.675,Z 150.000,A 0.000,B 0.000,C 180.000,E1 0.000} C_DIS
LIN {X -230.289,Y 35.867,Z 150.000,A 0.000,B 0.000,C 180.000,E1 0.000} C_DIS
LIN {X -231.830,Y 23.963,Z 150.000,A 0.000,B 0.000,C 180.000,E1 0.000} C_DIS
LIN {X -232.757,Y 11.999,Z 150.000,A 0.000,B 0.000,C 180.000,E1 0.000} C_DIS
LIN {X -233.065,Y 0.000,Z 150.000,A 0.000,B 0.000,C 180.000,E1 0.000} C_DIS
LIN {X -232.757,Y -11.999,Z 150.000,A 0.000,B 0.000,C 180.000,E1 0.000} C_DIS
LIN {X -231.830,Y -23.965,Z 150.000,A 0.000,B 0.000,C 180.000,E1 0.000} C_DIS
LIN {X -231.354,Y -27.651,Z 150.000,A 0.000,B 0.000,C 180.000,E1 0.000} C_DIS
LIN {X -230.289,Y -35.866,Z 150.000,A 0.000,B 0.000,C 180.000,E1 0.000} C_DIS
LIN {X -228.138,Y -47.675,Z 150.000,A 0.000,B 0.000,C 180.000,E1 0.000} C_DIS
LIN {X -225.381,Y -59.355,Z 150.000,A 0.000,B 0.000,C 180.000,E1 0.000} C_DIS
LIN {X -222.027,Y -70.878,Z 150.000,A 0.000,B 0.000,C 180.000,E1 0.000} C_DIS
LIN {X -218.083,Y -82.214,Z 150.000,A 0.000,B 0.000,C 180.000,E1 0.000} C_DIS
LIN {X -213.562,Y -93.332,Z 150.000,A 0.000,B 0.000,C 180.000,E1 0.000} C_DIS
LIN {X -208.475,Y -104.200,Z 150.000,A 0.000,B 0.000,C 180.000,E1 0.000} C_DIS
LIN {X -202.832,Y -114.796,Z 150.000,A 0.000,B 0.000,C 180.000,E1 0.000} C_DIS
LIN {X -196.655,Y -125.086,Z 150.000,A 0.000,B 0.000,C 180.000,E1 0.000} C_DIS
LIN {X -189.955,Y -135.043,Z 150.000,A 0.000,B 0.000,C 180.000,E1 0.000} C_DIS
LIN {X -182.751,Y -144.643,Z 150.000,A 0.000,B 0.000,C 180.000,E1 0.000} C_DIS
LIN {X -175.063,Y -153.859,Z 150.000,A 0.000,B 0.000,C 180.000,E1 0.000} C_DIS
LIN {X -166.911,Y -162.666,Z 150.000,A 0.000,B 0.000,C 180.000,E1 0.000} C_DIS
LIN {X -158.316,Y -171.043,Z 150.000,A 0.000,B 0.000,C 180.000,E1 0.000} C_DIS
LIN {X -149.299,Y -178.967,Z 150.000,A 0.000,B 0.000,C 180.000,E1 0.000} C_DIS
LIN {X -139.889,Y -186.416,Z 150.000,A 0.000,B 0.000,C 180.000,E1 0.000} C_DIS
LIN {X -130.108,Y -193.369,Z 150.000,A 0.000,B 0.000,C 180.000,E1 0.000} C_DIS
LIN {X -119.981,Y -199.810,Z 150.000,A 0.000,B 0.000,C 180.000,E1 0.000} C_DIS
LIN {X -109.536,Y -205.722,Z 150.000,A 0.000,B 0.000,C 180.000,E1 0.000} C_DIS
LIN {X -98.800,Y -211.088,Z 150.000,A 0.000,B 0.000,C 180.000,E1 0.000} C_DIS
LIN {X -87.802,Y -215.893,Z 150.000,A 0.000,B 0.000,C 180.000,E1 0.000} C_DIS
LIN {X -76.572,Y -220.127,Z 150.000,A 0.000,B 0.000,C 180.000,E1 0.000} C_DIS
LIN {X -65.137,Y -223.777,Z 150.000,A 0.000,B 0.000,C 180.000,E1 0.000} C_DIS
LIN {X -53.532,Y -226.835,Z 150.000,A 0.000,B 0.000,C 180.000,E1 0.000} C_DIS
LIN {X -41.784,Y -229.289,Z 150.000,A 0.000,B 0.000,C 180.000,E1 0.000} C_DIS
LIN {X -29.924,Y -231.137,Z 150.000,A 0.000,B 0.000,C 180.000,E1 0.000} C_DIS
LIN {X -17.987,Y -232.371,Z 150.000,A 0.000,B 0.000,C 180.000,E1 0.000} C_DIS
LIN {X -6.001,Y -232.988,Z 150.000,A 0.000,B 0.000,C 180.000,E1 0.000} C_DIS
LIN {X 6.001,Y -232.988,Z 150.000,A 0.000,B 0.000,C 180.000,E1 0.000} C_DIS
LIN {X 17.987,Y -232.371,Z 150.000,A 0.000,B 0.000,C 180.000,E1 0.000} C_DIS
LIN {X 29.924,Y -231.137,Z 150.000,A 0.000,B 0.000,C 180.000,E1 0.000} C_DIS
LIN {X 41.784,Y -229.289,Z 150.000,A 0.000,B 0.000,C 180.000,E1 0.000} C_DIS
LIN {X 53.532,Y -226.835,Z 150.000,A 0.000,B 0.000,C 180.000,E1 0.000} C_DIS
LIN {X 65.137,Y -223.777,Z 150.000,A 0.000,B 0.000,C 180.000,E1 0.000} C_DIS
LIN {X 76.572,Y -220.127,Z 150.000,A 0.000,B 0.000,C 180.000,E1 0.000} C_DIS
LIN {X 87.802,Y -215.893,Z 150.000,A 0.000,B 0.000,C 180.000,E1 0.000} C_DIS
LIN {X 98.800,Y -211.088,Z 150.000,A 0.000,B 0.000,C 180.000,E1 0.000} C_DIS
LIN {X 109.536,Y -205.722,Z 150.000,A 0.000,B 0.000,C 180.000,E1 0.000} C_DIS
LIN {X 119.981,Y -199.810,Z 150.000,A 0.000,B 0.000,C 180.000,E1 0.000} C_DIS
LIN {X 130.108,Y -193.369,Z 150.000,A 0.000,B 0.000,C 180.000,E1 0.000} C_DIS
LIN {X 139.889,Y -186.416,Z 150.000,A 0.000,B 0.000,C 180.000,E1 0.000} C_DIS
LIN {X 149.299,Y -178.967,Z 150.000,A 0.000,B 0.000,C 180.000,E1 0.000} C_DIS
LIN {X 158.316,Y -171.043,Z 150.000,A 0.000,B 0.000,C 180.000,E1 0.000} C_DIS
LIN {X 166.911,Y -162.666,Z 150.000,A 0.000,B 0.000,C 180.000,E1 0.000} C_DIS
LIN {X 175.063,Y -153.859,Z 150.000,A 0.000,B 0.000,C 180.000,E1 0.000} C_DIS
LIN {X 182.751,Y -144.643,Z 150.000,A 0.000,B 0.000,C 180.000,E1 0.000} C_DIS
LIN {X 189.955,Y -135.043,Z 150.000,A 0.000,B 0.000,C 180.000,E1 0.000} C_DIS
LIN {X 196.655,Y -125.086,Z 150.000,A 0.000,B 0.000,C 180.000,E1 0.000} C_DIS
LIN {X 202.832,Y -114.796,Z 150.000,A 0.000,B 0.000,C 180.000,E1 0.000} C_DIS
LIN {X 208.475,Y -104.200,Z 150.000,A 0.000,B 0.000,C 180.000,E1 0.000} C_DIS
LIN {X 213.562,Y -93.332,Z 150.000,A 0.000,B 0.000,C 180.000,E1 0.000} C_DIS
LIN {X 218.084,Y -82.213,Z 150.000,A 0.000,B 0.000,C 180.000,E1 0.000} C_DIS
LIN {X 222.026,Y -70.879,Z 150.000,A 0.000,B 0.000,C 180.000,E1 0.000} C_DIS
LIN {X 225.381,Y -59.355,Z 150.000,A 0.000,B 0.000,C 180.000,E1 0.000} C_DIS
LIN {X 228.138,Y -47.675,Z 150.000,A 0.000,B 0.000,C 180.000,E1 0.000} C_DIS
LIN {X 230.289,Y -35.867,Z 150.000,A 0.000,B 0.000,C 180.000,E1 0.000} C_DIS
LIN {X 231.830,Y -23.963,Z 150.000,A 0.000,B 0.000,C 180.000,E1 0.000} C_DIS
LIN {X 232.757,Y -11.999,Z 150.000,A 0.000,B 0.000,C 180.000,E1 0.000} C_DIS
LIN {X 233.065,Y 0.000,Z 150.000,A 0.000,B 0.000,C 180.000,E1 0.000} C_DIS
LIN {X 232.757,Y 11.999,Z 150.000,A 0.000,B 0.000,C 180.000,E1 0.000} C_DIS
LIN {X 231.830,Y 23.965,Z 150.000,A 0.000,B 0.000,C 180.000,E1 0.000} C_DIS
LIN {X 230.289,Y 35.866,Z 150.000,A 0.000,B 0.000,C 180.000,E1 0.000} C_DIS
LIN {X 228.138,Y 47.675,Z 150.000,A 0.000,B 0.000,C 180.000,E1 0.000} C_DIS
LIN {X 225.381,Y 59.355,Z 150.000,A 0.000,B 0.000,C 180.000,E1 0.000} C_DIS
LIN {X 222.027,Y 70.878,Z 150.000,A 0.000,B 0.000,C 180.000,E1 0.000} C_DIS
LIN {X 218.083,Y 82.214,Z 150.000,A 0.000,B 0.000,C 180.000,E1 0.000} C_DIS
LIN {X 213.562,Y 93.332,Z 150.000,A 0.000,B 0.000,C 180.000,E1 0.000} C_DIS
LIN {X 208.475,Y 104.200,Z 150.000,A 0.000,B 0.000,C 180.000,E1 0.000} C_DIS
LIN {X 202.832,Y 114.796,Z 150.000,A 0.000,B 0.000,C 180.000,E1 0.000} C_DIS
LIN {X 196.655,Y 125.086,Z 150.000,A 0.000,B 0.000,C 180.000,E1 0.000} C_DIS
LIN {X 189.955,Y 135.043,Z 150.000,A 0.000,B 0.000,C 180.000,E1 0.000} C_DIS
LIN {X 182.751,Y 144.643,Z 150.000,A 0.000,B 0.000,C 180.000,E1 0.000} C_DIS
LIN {X 175.063,Y 153.859,Z 150.000,A 0.000,B 0.000,C 180.000,E1 0.000} C_DIS
LIN {X 166.911,Y 162.666,Z 150.000,A 0.000,B 0.000,C 180.000,E1 0.000} C_DIS
LIN {X 158.316,Y 171.043,Z 150.000,A 0.000,B 0.000,C 180.000,E1 0.000} C_DIS
LIN {X 149.299,Y 178.967,Z 150.000,A 0.000,B 0.000,C 180.000,E1 0.000} C_DIS
LIN {X 139.889,Y 186.416,Z 150.000,A 0.000,B 0.000,C 180.000,E1 0.000} C_DIS
LIN {X 130.108,Y 193.369,Z 150.000,A 0.000,B 0.000,C 180.000,E1 0.000} C_DIS
;rapid-leaky
$VEL.CP=0.3
LIN {X 84.633,Y 197.897,Z 150.000,A 0.000,B 0.000,C 180.000,E1 0.000} C_DIS
;bead-sparse_infill
$VEL.CP=0.63
LIN {X 197.949,Y 84.581,Z 150.000,A 0.000,B 0.000,C 180.000,E1 0.000} C_DIS
LIN {X 201.459,Y 75.948,Z 150.000,A 0.000,B 0.000,C 180.000,E1 0.000} C_DIS
LIN {X 205.102,Y 65.475,Z 150.000,A 0.000,B 0.000,C 180.000,E1 0.000} C_DIS
LIN {X 208.201,Y 54.831,Z 150.000,A 0.000,B 0.000,C 180.000,E1 0.000} C_DIS
LIN {X 210.747,Y 44.041,Z 150.000,A 0.000,B 0.000,C 180.000,E1 0.000} C_DIS
LIN {X 212.735,Y 33.132,Z 150.000,A 0.000,B 0.000,C 180.000,E1 0.000} C_DIS
LIN {X 214.159,Y 22.138,Z 150.000,A 0.000,B 0.000,C 180.000,E1 0.000} C_DIS
LIN {X 215.014,Y 11.084,Z 150.000,A 0.000,B 0.000,C 180.000,E1 0.000} C_DIS
LIN {X 215.299,Y 0.000,Z 150.000,A 0.000,B 0.000,C 180.000,E1 0.000} C_DIS
LIN {X 215.014,Y -11.084,Z 150.000,A 0.000,B 0.000,C 180.000,E1 0.000} C_DIS
LIN {X 214.159,Y -22.136,Z 150.000,A 0.000,B 0.000,C 180.000,E1 0.000} C_DIS
LIN {X 212.734,Y -33.133,Z 150.000,A 0.000,B 0.000,C 180.000,E1 0.000} C_DIS
LIN {X 210.747,Y -44.041,Z 150.000,A 0.000,B 0.000,C 180.000,E1 0.000} C_DIS
LIN {X 208.201,Y -54.831,Z 150.000,A 0.000,B 0.000,C 180.000,E1 0.000} C_DIS
LIN {X 205.102,Y -65.476,Z 150.000,A 0.000,B 0.000,C 180.000,E1 0.000} C_DIS
LIN {X 201.470,Y -75.918,Z 150.000,A 0.000,B 0.000,C 180.000,E1 0.000} C_DIS
LIN {X -75.863,Y 201.414,Z 150.000,A 0.000,B 0.000,C 180.000,E1 0.000} C_DIS
LIN {X -81.109,Y 199.436,Z 150.000,A 0.000,B 0.000,C 180.000,E1 0.000} C_DIS
LIN {X -91.269,Y 194.997,Z 150.000,A 0.000,B 0.000,C 180.000,E1 0.000} C_DIS
LIN {X -101.186,Y 190.040,Z 150.000,A 0.000,B 0.000,C 180.000,E1 0.000} C_DIS
LIN {X -110.835,Y 184.579,Z 150.000,A 0.000,B 0.000,C 180.000,E1 0.000} C_DIS
LIN {X -120.191,Y 178.629,Z 150.000,A 0.000,B 0.000,C 180.000,E1 0.000} C_DIS
LIN {X -129.226,Y 172.206,Z 150.000,A 0.000,B 0.000,C 180.000,E1 0.000} C_DIS
LIN {X -137.918,Y 165.325,Z 150.000,A 0.000,B 0.000,C 180.000,E1 0.000} C_DIS
LIN {X -146.248,Y 158.004,Z 150.000,A 0.000,B 0.000,C 180.000,E1 0.000} C_DIS
LIN {X -154.188,Y 150.266,Z 150.000,A 0.000,B 0.000,C 180.000,E1 0.000} C_DIS
LIN {X -161.718,Y 142.131,Z 150.000,A 0.000,B 0.000,C 180.000,E1 0.000} C_DIS
LIN {X -167.103,Y 135.676,Z 150.000,A 0.000,B 0.000,C 180.000,E1 0.000} C_DIS
LIN {X 135.675,Y -167.101,Z 150.000,A 0.000,B 0.000,C 180.000,E1 0.000} C_DIS
LIN {X 129.226,Y -172.206,Z 150.000,A 0.000,B 0.000,C 180.000,E1 0.000} C_DIS
LIN {X 120.191,Y -178.629,Z 150.000,A 0.000,B 0.000,C 180.000,E1 0.000} C_DIS
LIN {X 110.835,Y -184.579,Z 150.000,A 0.000,B 0.000,C 180.000,E1 0.000} C_DIS
LIN {X 101.186,Y -190.040,Z 150.000,A 0.000,B 0.000,C 180.000,E1 0.000} C_DIS
LIN {X 91.269,Y -194.997,Z 150.000,A 0.000,B 0.000,C 180.000,E1 0.000} C_DIS
LIN {X 81.109,Y -199.436,Z 150.000,A 0.000,B 0.000,C 180.000,E1 0.000} C_DIS
LIN {X 70.735,Y -203.348,Z 150.000,A 0.000,B 0.000,C 180.000,E1 0.000} C_DIS
LIN {X 60.172,Y -206.720,Z 150.000,A 0.000,B 0.000,C 180.000,E1 0.000} C_DIS
LIN {X 49.451,Y -209.544,Z 150.000,A 0.000,B 0.000,C 180.000,E1 0.000} C_DIS
LIN {X 38.599,Y -211.811,Z 150.000,A 0.000,B 0.000,C 180.000,E1 0.000} C_DIS
LIN {X 27.642,Y -213.518,Z 150.000,A 0.000,B 0.000,C 180.000,E1 0.000} C_DIS
LIN {X 25.351,Y -213.755,Z 150.000,A 0.000,B 0.000,C 180.000,E1 0.000} C_DIS
LIN {X -213.744,Y 25.340,Z 150.000,A 0.000,B 0.000,C 180.000,E1 0.000} C_DIS
;rapid-leaky
$VEL.CP=0.3
LIN {X 55.730,Y -236.147,Z 160.000,A 0.000,B 0.000,C 180.000,E1 0.000} C_DIS
;bead-perimeter_outer
$VEL.CP=0.62
LIN {X 67.813,Y -232.965,Z 160.000,A 0.000,B 0.000,C 180.000,E1 0.000} C_DIS
LIN {X 79.716,Y -229.165,Z 160.000,A 0.000,B 0.000,C 180.000,E1 0.000} C_DIS
LIN {X 91.406,Y -224.757,Z 160.000,A 0.000,B 0.000,C 180.000,E1 0.000} C_DIS
LIN {X 102.856,Y -219.754,Z 160.000,A 0.000,B 0.000,C 180.000,E1 0.000} C_DIS
LIN {X 114.032,Y -214.167,Z 160.000,A 0.000,B 0.000,C 180.000,E1 0.000} C_DIS
LIN {X 124.906,Y -208.014,Z 160.000,A 0.000,B 0.000,C 180.000,E1 0.000} C_DIS
LIN {X 135.448,Y -201.308,Z 160.000,A 0.000,B 0.000,C 180.000,E1 0.000} C_DIS
LIN {X 145.633,Y -194.068,Z 160.000,A 0.000,B 0.000,C 180.000,E1 0.000} C_DIS
LIN {X 155.430,Y -186.314,Z 160.000,A 0.000,B 0.000,C 180.000,E1 0.000} C_DIS
LIN {X 164.813,Y -178.065,Z 160.000,A 0.000,B 0.000,C 180.000,E1 0.000} C_DIS
LIN {X 173.763,Y -169.344,Z 160.000,A 0.000,B 0.000,C 180.000,E1 0.000} C_DIS
LIN {X 182.250,Y -160.175,Z 160.000,A 0.000,B 0.000,C 180.000,E1 0.000} C_DIS
LIN {X 190.254,Y -150.581,Z 160.000,A 0.000,B 0.000,C 180.000,E1 0.000} C_DIS
LIN {X 197.753,Y -140.587,Z 160.000,A 0.000,B 0.000,C 180.000,E1 0.000} C_DIS
LIN {X 204.729,Y -130.221,Z 160.000,A 0.000,B 0.000,C 180.000,E1 0.000} C_DIS
LIN {X 211.160,Y -119.508,Z 160.000,A 0.000,B 0.000,C 180.000,E1 0.000} C_DIS
LIN {X 217.032,Y -108.480,Z 160.000,A 0.000,B 0.000,C 180.000,E1 0.000} C_DIS
LIN {X 222.329,Y -97.163,Z 160.000,A 0.000,B 0.000,C 180.000,E1 0.000} C_DIS
LIN {X 227.036,Y -85.589,Z 160.000,A 0.000,B 0.000,C 180.000,E1 0.000} C_DIS
LIN {X 231.141,Y -73.789,Z 160.000,A 0.000,B 0.000,C 180.000,E1 0.000} C_DIS
LIN {X 234.633,Y -61.792,Z 160.000,A 0.000,B 0.000,C 180.000,E1 0.000} C_DIS
LIN {X 237.503,Y -49.632,Z 160.000,A 0.000,B 0.000,C 180.000,E1 0.000} C_DIS
LIN {X 239.744,Y -37.339,Z 160.000,A 0.000,B 0.000,C 180.000,E1 0.000} C_DIS
LIN {X 241.347,Y -24.948,Z 160.000,A 0.000,B 0.000,C 180.000,E1 0.000} C_DIS
LIN {X 242.312,Y -12.490,Z 160.000,A 0.000,B 0.000,C 180.000,E1 0.000} C_DIS
LIN {X 242.633,Y 0.000,Z 160.000,A 0.000,B 0.000,C 180.000,E1 0.000} C_DIS
LIN {X 242.312,Y 12.490,Z 160.000,A 0.000,B 0.000,C 180.000,E1 0.000} C_DIS
LIN {X 241.347,Y 24.948,Z 160.000,A 0.000,B 0.000,C 180.000,E1 0.000} C_DIS
LIN {X 239.744,Y 37.339,Z 160.000,A 0.000,B 0.000,C 180.000,E1 0.000} C_DIS
LIN {X 237.503,Y 49.632,Z 160.000,A 0.000,B 0.000,C 180.000,E1 0.000} C_DIS
LIN {X 234.633,Y 61.792,Z 160.000,A 0.000,B 0.000,C 180.000,E1 0.000} C_DIS
LIN {X 231.141,Y 73.789,Z 160.000,A 0.000,B 0.000,C 180.000,E1 0.000} C_DIS
LIN {X 227.036,Y 85.589,Z 160.000,A 0.000,B 0.000,C 180.000,E1 0.000} C_DIS
LIN {X 222.328,Y 97.165,Z 160.000,A 0.000,B 0.000,C 180.000,E1 0.000} C_DIS
LIN {X 217.032,Y 108.480,Z 160.000,A 0.000,B 0.000,C 180.000,E1 0.000} C_DIS
LIN {X 211.160,Y 119.508,Z 160.000,A 0.000,B 0.000,C 180.000,E1 0.000} C_DIS
LIN {X 204.729,Y 130.221,Z 160.000,A 0.000,B 0.000,C 180.000,E1 0.000} C_DIS
LIN {X 197.753,Y 140.587,Z 160.000,A 0.000,B 0.000,C 180.000,E1 0.000} C_DIS
LIN {X 190.254,Y 150.581,Z 160.000,A 0.000,B 0.000,C 180.000,E1 0.000} C_DIS
LIN {X 182.250,Y 160.175,Z 160.000,A 0.000,B 0.000,C 180.000,E1 0.000} C_DIS
LIN {X 173.763,Y 169.344,Z 160.000,A 0.000,B 0.000,C 180.000,E1 0.000} C_DIS
LIN {X 164.813,Y 178.065,Z 160.000,A 0.000,B 0.000,C 180.000,E1 0.000} C_DIS
LIN {X 155.430,Y 186.314,Z 160.000,A 0.000,B 0.000,C 180.000,E1 0.000} C_DIS
LIN {X 145.633,Y 194.068,Z 160.000,A 0.000,B 0.000,C 180.000,E1 0.000} C_DIS
LIN {X 135.448,Y 201.308,Z 160.000,A 0.000,B 0.000,C 180.000,E1 0.000} C_DIS
LIN {X 124.906,Y 208.014,Z 160.000,A 0.000,B 0.000,C 180.000,E1 0.000} C_DIS
LIN {X 114.032,Y 214.167,Z 160.000,A 0.000,B 0.000,C 180.000,E1 0.000} C_DIS
LIN {X 102.856,Y 219.754,Z 160.000,A 0.000,B 0.000,C 180.000,E1 0.000} C_DIS
LIN {X 91.405,Y 224.758,Z 160.000,A 0.000,B 0.000,C 180.000,E1 0.000} C_DIS
LIN {X 79.716,Y 229.165,Z 160.000,A 0.000,B 0.000,C 180.000,E1 0.000} C_DIS
LIN {X 67.813,Y 232.965,Z 160.000,A 0.000,B 0.000,C 180.000,E1 0.000} C_DIS
LIN {X 55.730,Y 236.147,Z 160.000,A 0.000,B 0.000,C 180.000,E1 0.000} C_DIS
LIN {X 43.500,Y 238.702,Z 160.000,A 0.000,B 0.000,C 180.000,E1 0.000} C_DIS
LIN {X 31.153,Y 240.625,Z 160.000,A 0.000,B 0.000,C 180.000,E1 0.000} C_DIS
LIN {X 18.725,Y 241.909,Z 160.000,A 0.000,B 0.000,C 180.000,E1 0.000} C_DIS
LIN {X 6.247,Y 242.553,Z 160.000,A 0.000,B 0.000,C 180.000,E1 0.000} C_DIS
LIN {X -6.247,Y 242.553,Z 160.000,A 0.000,B 0.000,C 180.000,E1 0.000} C_DIS
LIN {X -18.725,Y 241.909,Z 160.000,A 0.000,B 0.000,C 180.000,E1 0.000} C_DIS
LIN {X -31.153,Y 240.625,Z 160.000,A 0.000,B 0.000,C 180.000,E1 0.000} C_DIS
LIN {X -43.500,Y 238.702,Z 160.000,A 0.000,B 0.000,C 180.000,E1 0.000} C_DIS
LIN {X -55.730,Y 236.147,Z 160.000,A 0.000,B 0.000,C 180.000,E1 0.000} C_DIS
LIN {X -67.813,Y 232.965,Z 160.000,A 0.000,B 0.000,C 180.000,E1 0.000} C_DIS
LIN {X -79.716,Y 229.165,Z 160.000,A 0.000,B 0.000,C 180.000,E1 0.000} C_DIS
LIN {X -91.406,Y 224.757,Z 160.000,A 0.000,B 0.000,C 180.000,E1 0.000} C_DIS
LIN {X -102.856,Y 219.754,Z 160.000,A 0.000,B 0.000,C 180.000,E1 0.000} C_DIS
LIN {X -114.032,Y 214.167,Z 160.000,A 0.000,B 0.000,C 180.000,E1 0.000} C_DIS
LIN {X -124.906,Y 208.014,Z 160.000,A 0.000,B 0.000,C 180.000,E1 0.000} C_DIS
LIN {X -135.448,Y 201.308,Z 160.000,A 0.000,B 0.000,C 180.000,E1 0.000} C_DIS
LIN {X -145.633,Y 194.068,Z 160.000,A 0.000,B 0.000,C 180.000,E1 0.000} C_DIS
LIN {X -155.430,Y 186.314,Z 160.000,A 0.000,B 0.000,C 180.000,E1 0.000} C_DIS
LIN {X -164.813,Y 178.065,Z 160.000,A 0.000,B 0.000,C 180.000,E1 0.000} C_DIS
LIN {X -173.763,Y 169.344,Z 160.000,A 0.000,B 0.000,C 180.000,E1 0.000} C_DIS
LIN {X -182.250,Y 160.175,Z 160.000,A 0.000,B 0.000,C 180.000,E1 0.000} C_DIS
LIN {X -190.254,Y 150.581,Z 160.000,A 0.000,B 0.000,C 180.000,E1 0.000} C_DIS
LIN {X -197.753,Y 140.587,Z 160.000,A 0.000,B 0.000,C 180.000,E1 0.000} C_DIS
LIN {X -204.729,Y 130.221,Z 160.000,A 0.000,B 0.000,C 180.000,E1 0.000} C_DIS
LIN {X -211.160,Y 119.508,Z 160.000,A 0.000,B 0.000,C 180.000,E1 0.000} C_DIS
LIN {X -217.032,Y 108.480,Z 160.000,A 0.000,B 0.000,C 180.000,E1 0.000} C_DIS
LIN {X -222.329,Y 97.163,Z 160.000,A 0.000,B 0.000,C 180.000,E1 0.000} C_DIS
LIN {X -227.036,Y 85.589,Z 160.000,A 0.000,B 0.000,C 180.000,E1 0.000} C_DIS
LIN {X -231.141,Y 73.789,Z 160.000,A 0.000,B 0.000,C 180.000,E1 0.000} C_DIS
LIN {X -234.633,Y 61.792,Z 160.000,A 0.000,B 0.000,C 180.000,E1 0.000} C_DIS
LIN {X -237.503,Y 49.632,Z 160.000,A 0.000,B 0.000,C 180.000,E1 0.000} C_DIS
LIN {X -239.744,Y 37.339,Z 160.000,A 0.000,B 0.000,C 180.000,E1 0.000} C_DIS
LIN {X -241.347,Y 24.948,Z 160.000,A 0.000,B 0.000,C 180.000,E1 0.000} C_DIS
LIN {X -242.312,Y 12.490,Z 160.000,A 0.000,B 0.000,C 180.000,E1 0.000} C_DIS
LIN {X -242.633,Y 0.000,Z 160.000,A 0.000,B 0.000,C 180.000,E1 0.000} C_DIS
LIN {X -242.312,Y -12.490,Z 160.000,A 0.000,B 0.000,C 180.000,E1 0.000} C_DIS
LIN {X -241.347,Y -24.948,Z 160.000,A 0.000,B 0.000,C 180.000,E1 0.000} C_DIS
LIN {X -239.744,Y -37.339,Z 160.000,A 0.000,B 0.000,C 180.000,E1 0.000} C_DIS
LIN {X -237.503,Y -49.632,Z 160.000,A 0.000,B 0.000,C 180.000,E1 0.000} C_DIS
LIN {X -234.633,Y -61.792,Z 160.000,A 0.000,B 0.000,C 180.000,E1 0.000} C_DIS
LIN {X -231.141,Y -73.789,Z 160.000,A 0.000,B 0.000,C 180.000,E1 0.000} C_DIS
LIN {X -227.036,Y -85.589,Z 160.000,A 0.000,B 0.000,C 180.000,E1 0.000} C_DIS
LIN {X -222.328,Y -97.165,Z 160.000,A 0.000,B 0.000,C 180.000,E1 0.000} C_DIS
LIN {X -217.032,Y -108.480,Z 160.000,A 0.000,B 0.000,C 180.000,E1 0.000} C_DIS
LIN {X -211.160,Y -119.508,Z 160.000,A 0.000,B 0.000,C 180.000,E1 0.000} C_DIS
LIN {X -204.729,Y -130.221,Z 160.000,A 0.000,B 0.000,C 180.000,E1 0.000} C_DIS
LIN {X -197.753,Y -140.587,Z 160.000,A 0.000,B 0.000,C 180.000,E1 0.000} C_DIS
LIN {X -190.254,Y -150.581,Z 160.000,A 0.000,B 0.000,C 180.000,E1 0.000} C_DIS
LIN {X -182.250,Y -160.175,Z 160.000,A 0.000,B 0.000,C 180.000,E1 0.000} C_DIS
LIN {X -173.763,Y -169.344,Z 160.000,A 0.000,B 0.000,C 180.000,E1 0.000} C_DIS
LIN {X -164.813,Y -178.065,Z 160.000,A 0.000,B 0.000,C 180.000,E1 0.000} C_DIS
LIN {X -155.430,Y -186.314,Z 160.000,A 0.000,B 0.000,C 180.000,E1 0.000} C_DIS
LIN {X -145.633,Y -194.068,Z 160.000,A 0.000,B 0.000,C 180.000,E1 0.000} C_DIS
LIN {X -135.448,Y -201.308,Z 160.000,A 0.000,B 0.000,C 180.000,E1 0.000} C_DIS
LIN {X -124.906,Y -208.014,Z 160.000,A 0.000,B 0.000,C 180.000,E1 0.000} C_DIS
LIN {X -114.032,Y -214.167,Z 160.000,A 0.000,B 0.000,C 180.000,E1 0.000} C_DIS
LIN {X -102.856,Y -219.754,Z 160.000,A 0.000,B 0.000,C 180.000,E1 0.000} C_DIS
LIN {X -91.405,Y -224.758,Z 160.000,A 0.000,B 0.000,C 180.000,E1 0.000} C_DIS
LIN {X -79.716,Y -229.165,Z 160.000,A 0.000,B 0.000,C 180.000,E1 0.000} C_DIS
LIN {X -67.813,Y -232.965,Z 160.000,A 0.000,B 0.000,C 180.000,E1 0.000} C_DIS
LIN {X -55.730,Y -236.147,Z 160.000,A 0.000,B 0.000,C 180.000,E1 0.000} C_DIS
LIN {X -43.500,Y -238.702,Z 160.000,A 0.000,B 0.000,C 180.000,E1 0.000} C_DIS
LIN {X -31.153,Y -240.625,Z 160.000,A 0.000,B 0.000,C 180.000,E1 0.000} C_DIS
LIN {X -18.725,Y -241.909,Z 160.000,A 0.000,B 0.000,C 180.000,E1 0.000} C_DIS
LIN {X -6.247,Y -242.553,Z 160.000,A 0.000,B 0.000,C 180.000,E1 0.000} C_DIS
LIN {X 6.247,Y -242.553,Z 160.000,A 0.000,B 0.000,C 180.000,E1 0.000} C_DIS
LIN {X 18.725,Y -241.909,Z 160.000,A 0.000,B 0.000,C 180.000,E1 0.000} C_DIS
LIN {X 31.153,Y -240.625,Z 160.000,A 0.000,B 0.000,C 180.000,E1 0.000} C_DIS
LIN {X 43.500,Y -238.702,Z 160.000,A 0.000,B 0.000,C 180.000,E1 0.000} C_DIS
LIN {X 55.730,Y -236.147,Z 160.000,A 0.000,B 0.000,C 180.000,E1 0.000} C_DIS
;rapid-leaky
$VEL.CP=0.3
LIN {X 52.160,Y -221.018,Z 160.000,A 0.000,B 0.000,C 180.000,E1 0.000} C_DIS
;bead-perimeter_inner
$VEL.CP=0.62
LIN {X 63.468,Y -218.039,Z 160.000,A 0.000,B 0.000,C 180.000,E1 0.000} C_DIS
LIN {X 74.608,Y -214.483,Z 160.000,A 0.000,B 0.000,C 180.000,E1 0.000} C_DIS
LIN {X 85.550,Y -210.357,Z 160.000,A 0.000,B 0.000,C 180.000,E1 0.000} C_DIS
LIN {X 96.266,Y -205.675,Z 160.000,A 0.000,B 0.000,C 180.000,E1 0.000} C_DIS
LIN {X 106.726,Y -200.446,Z 160.000,A 0.000,B 0.000,C 180.000,E1 0.000} C_DIS
LIN {X 116.903,Y -194.686,Z 160.000,A 0.000,B 0.000,C 180.000,E1 0.000} C_DIS
LIN {X 126.770,Y -188.410,Z 160.000,A 0.000,B 0.000,C 180.000,E1 0.000} C_DIS
LIN {X 136.302,Y -181.634,Z 160.000,A 0.000,B 0.000,C 180.000,E1 0.000} C_DIS
LIN {X 145.471,Y -174.377,Z 160.000,A 0.000,B 0.000,C 180.000,E1 0.000} C_DIS
LIN {X 154.254,Y -166.657,Z 160.000,A 0.000,B 0.000,C 180.000,E1 0.000} C_DIS
LIN {X 162.631,Y -158.494,Z 160.000,A 0.000,B 0.000,C 180.000,E1 0.000} C_DIS
LIN {X 170.574,Y -149.912,Z 160.000,A 0.000,B 0.000,C 180.000,E1 0.000} C_DIS
LIN {X 178.065,Y -140.933,Z 160.000,A 0.000,B 0.000,C 180.000,E1 0.000} C_DIS
LIN {X 185.084,Y -131.580,Z 160.000,A 0.000,B 0.000,C 180.000,E1 0.000} C_DIS
LIN {X 191.612,Y -121.878,Z 160.000,A 0.000,B 0.000,C 180.000,E1 0.000} C_DIS
LIN {X 197.631,Y -111.853,Z 160.000,A 0.000,B 0.000,C 180.000,E1 0.000} C_DIS
LIN {X 203.127,Y -101.530,Z 160.000,A 0.000,B 0.000,C 180.000,E1 0.000} C_DIS
LIN {X 208.084,Y -90.938,Z 160.000,A 0.000,B 0.000,C 180.000,E1 0.000} C_DIS
LIN {X 212.491,Y -80.105,Z 160.000,A 0.000,B 0.000,C 180.000,E1 0.000} C_DIS
LIN {X 216.333,Y -69.061,Z 160.000,A 0.000,B 0.000,C 180.000,E1 0.000} C_DIS
LIN {X 219.601,Y -57.833,Z 160.000,A 0.000,B 0.000,C 180.000,E1 0.000} C_DIS
LIN {X 222.287,Y -46.452,Z 160.000,A 0.000,B 0.000,C 180.000,E1 0.000} C_DIS
LIN {X 224.384,Y -34.947,Z 160.000,A 0.000,B 0.000,C 180.000,E1 0.000} C_DIS
LIN {X 225.884,Y -23.350,Z 160.000,A 0.000,B 0.000,C 180.000,E1 0.000} C_DIS
LIN {X 226.787,Y -11.690,Z 160.000,A 0.000,B 0.000,C 180.000,E1 0.000} C_DIS
LIN {X 227.088,Y 0.000,Z 160.000,A 0.000,B 0.000,C 180.000,E1 0.000} C_DIS
LIN {X 226.787,Y 11.690,Z 160.000,A 0.000,B 0.000,C 180.000,E1 0.000} C_DIS
LIN {X 225.884,Y 23.350,Z 160.000,A 0.000,B 0.000,C 180.000,E1 0.000} C_DIS
LIN {X 224.384,Y 34.947,Z 160.000,A 0.000,B 0.000,C 180.000,E1 0.000} C_DIS
LIN {X 222.287,Y 46.452,Z 160.000,A 0.000,B 0.000,C 180.000,E1 0.000} C_DIS
LIN {X 219.601,Y 57.833,Z 160.000,A 0.000,B 0.000,C 180.000,E1 0.000} C_DIS
LIN {X 216.333,Y 69.061,Z 160.000,A 0.000,B 0.000,C 180.000,E1 0.000} C_DIS
LIN {X 212.491,Y 80.105,Z 160.000,A 0.000,B 0.000,C 180.000,E1 0.000} C_DIS
LIN {X 208.083,Y 90.942,Z 160.000,A 0.000,B 0.000,C 180.000,E1 0.000} C_DIS
LIN {X 203.127,Y 101.530,Z 160.000,A 0.000,B 0.000,C 180.000,E1 0.000} C_DIS
LIN {X 197.631,Y 111.853,Z 160.000,A 0.000,B 0.000,C 180.000,E1 0.000} C_DIS
LIN {X 191.612,Y 121.878,Z 160.000,A 0.000,B 0.000,C 180.000,E1 0.000} C_DIS
LIN {X 185.084,Y 131.580,Z 160.000,A 0.000,B 0.000,C 180.000,E1 0.000} C_DIS
LIN {X 178.065,Y 140.933,Z 160.000,A 0.000,B 0.000,C 180.000,E1 0.000} C_DIS
LIN {X 170.574,Y 149.912,Z 160.000,A 0.000,B 0.000,C 180.000,E1 0.000} C_DIS
LIN {X 162.631,Y 158.494,Z 160.000,A 0.000,B 0.000,C 180.000,E1 0.000} C_DIS
LIN {X 154.254,Y 166.657,Z 160.000,A 0.000,B 0.000,C 180.000,E1 0.000} C_DIS
LIN {X 145.471,Y 174.377,Z 160.000,A 0.000,B 0.000,C 180.000,E1 0.000} C_DIS
LIN {X 136.302,Y 181.634,Z 160.000,A 0.000,B 0.000,C 180.000,E1 0.000} C_DIS
LIN {X 126.770,Y 188.410,Z 160.000,A 0.000,B 0.000,C 180.000,E1 0.000} C_DIS
LIN {X 116.903,Y 194.686,Z 160.000,A 0.000,B 0.000,C 180.000,E1 0.000} C_DIS
LIN {X 106.726,Y 200.446,Z 160.000,A 0.000,B 0.000,C 180.000,E1 0.000} C_DIS
LIN {X 96.266,Y 205.675,Z 160.000,A 0.000,B 0.000,C 180.000,E1 0.000} C_DIS
LIN {X 85.547,Y 210.359,Z 160.000,A 0.000,B 0.000,C 180.000,E1 0.000} C_DIS
LIN {X 74.609,Y 214.483,Z 160.000,A 0.000,B 0.000,C 180.000,E1 0.000} C_DIS
LIN {X 63.468,Y 218.039,Z 160.000,A 0.000,B 0.000,C 180.000,E1 0.000} C_DIS
LIN {X 52.160,Y 221.018,Z 160.000,A 0.000,B 0.000,C 180.000,E1 0.000} C_DIS
LIN {X 40.713,Y 223.409,Z 160.000,A 0.000,B 0.000,C 180.000,E1 0.000} C_DIS
LIN {X 29.158,Y 225.209,Z 160.000,A 0.000,B 0.000,C 180.000,E1 0.000} C_DIS
LIN {X 17.525,Y 226.411,Z 160.000,A 0.000,B 0.000,C 180.000,E1 0.000} C_DIS
LIN {X 5.846,Y 227.013,Z 160.000,A 0.000,B 0.000,C 180.000,E1 0.000} C_DIS
LIN {X -5.846,Y 227.013,Z 160.000,A 0.000,B 0.000,C 180.000,E1 0.000} C_DIS
LIN {X -17.525,Y 226.411,Z 160.000,A 0.000,B 0.000,C 180.000,E1 0.000} C_DIS
LIN {X -29.158,Y 225.209,Z 160.000,A 0.000,B 0.000,C 180.000,E1 0.000} C_DIS
LIN {X -40.713,Y 223.409,Z 160.000,A 0.000,B 0.000,C 180.000,E1 0.000} C_DIS
LIN {X -52.160,Y 221.018,Z 160.000,A 0.000,B 0.000,C 180.000,E1 0.000} C_DIS
LIN {X -63.468,Y 218.039,Z 160.000,A 0.000,B 0.000,C 180.000,E1 0.000} C_DIS
LIN {X -74.608,Y 214.483,Z 160.000,A 0.000,B 0.000,C 180.000,E1 0.000} C_DIS
LIN {X -85.550,Y 210.357,Z 160.000,A 0.000,B 0.000,C 180.000,E1 0.000} C_DIS
LIN {X -96.266,Y 205.675,Z 160.000,A 0.000,B 0.000,C 180.000,E1 0.000} C_DIS
LIN {X -106.726,Y 200.446,Z 160.000,A 0.000,B 0.000,C 180.000,E1 0.000} C_DIS
LIN {X -116.903,Y 194.686,Z 160.000,A 0.000,B 0.000,C 180.000,E1 0.000} C_DIS
LIN {X -126.770,Y 188.410,Z 160.000,A 0.000,B 0.000,C 180.000,E1 0.000} C_DIS
LIN {X -136.302,Y 181.634,Z 160.000,A 0.000,B 0.000,C 180.000,E1 0.000} C_DIS
LIN {X -145.471,Y 174.377,Z 160.000,A 0.000,B 0.000,C 180.000,E1 0.000} C_DIS
LIN {X -154.254,Y 166.657,Z 160.000,A 0.000,B 0.000,C 180.000,E1 0.000} C_DIS
LIN {X -162.631,Y 158.494,Z 160.000,A 0.000,B 0.000,C 180.000,E1 0.000} C_DIS
LIN {X -170.574,Y 149.912,Z 160.000,A 0.000,B 0.000,C 180.000,E1 0.000} C_DIS
LIN {X -178.065,Y 140.933,Z 160.000,A 0.000,B 0.000,C 180.000,E1 0.000} C_DIS
LIN {X -185.084,Y 131.580,Z 160.000,A 0.000,B 0.000,C 180.000,E1 0.000} C_DIS
LIN {X -191.612,Y 121.878,Z 160.000,A 0.000,B 0.000,C 180.000,E1 0.000} C_DIS
LIN {X -197.631,Y 111.853,Z 160.000,A 0.000,B 0.000,C 180.000,E1 0.000} C_DIS
LIN {X -203.127,Y 101.530,Z 160.000,A 0.000,B 0.000,C 180.000,E1 0.000} C_DIS
LIN {X -208.084,Y 90.938,Z 160.000,A 0.000,B 0.000,C 180.000,E1 0.000} C_DIS
LIN {X -212.491,Y 80.105,Z 160.000,A 0.000,B 0.000,C 180.000,E1 0.000} C_DIS
LIN {X -216.333,Y 69.061,Z 160.000,A 0.000,B 0.000,C 180.000,E1 0.000} C_DIS
LIN {X -219.601,Y 57.833,Z 160.000,A 0.000,B 0.000,C 180.000,E1 0.000} C_DIS
LIN {X -222.287,Y 46.452,Z 160.000,A 0.000,B 0.000,C 180.000,E1 0.000} C_DIS
LIN {X -224.384,Y 34.947,Z 160.000,A 0.000,B 0.000,C 180.000,E1 0.000} C_DIS
LIN {X -225.884,Y 23.350,Z 160.000,A 0.000,B 0.000,C 180.000,E1 0.000} C_DIS
LIN {X -226.787,Y 11.690,Z 160.000,A 0.000,B 0.000,C 180.000,E1 0.000} C_DIS
LIN {X -227.088,Y 0.000,Z 160.000,A 0.000,B 0.000,C 180.000,E1 0.000} C_DIS
LIN {X -226.787,Y -11.690,Z 160.000,A 0.000,B 0.000,C 180.000,E1 0.000} C_DIS
LIN {X -225.884,Y -23.350,Z 160.000,A 0.000,B 0.000,C 180.000,E1 0.000} C_DIS
LIN {X -224.384,Y -34.947,Z 160.000,A 0.000,B 0.000,C 180.000,E1 0.000} C_DIS
LIN {X -222.287,Y -46.452,Z 160.000,A 0.000,B 0.000,C 180.000,E1 0.000} C_DIS
LIN {X -219.601,Y -57.833,Z 160.000,A 0.000,B 0.000,C 180.000,E1 0.000} C_DIS
LIN {X -216.333,Y -69.061,Z 160.000,A 0.000,B 0.000,C 180.000,E1 0.000} C_DIS
LIN {X -212.491,Y -80.105,Z 160.000,A 0.000,B 0.000,C 180.000,E1 0.000} C_DIS
LIN {X -208.083,Y -90.942,Z 160.000,A 0.000,B 0.000,C 180.000,E1 0.000} C_DIS
LIN {X -203.127,Y -101.530,Z 160.000,A 0.000,B 0.000,C 180.000,E1 0.000} C_DIS
LIN {X -197.631,Y -111.853,Z 160.000,A 0.000,B 0.000,C 180.000,E1 0.000} C_DIS
LIN {X -191.612,Y -121.878,Z 160.000,A 0.000,B 0.000,C 180.000,E1 0.000} C_DIS
LIN {X -185.084,Y -131.580,Z 160.000,A 0.000,B 0.000,C 180.000,E1 0.000} C_DIS
LIN {X -178.065,Y -140.933,Z 160.000,A 0.000,B 0.000,C 180.000,E1 0.000} C_DIS
LIN {X -170.574,Y -149.912,Z 160.000,A 0.000,B 0.000,C 180.000,E1 0.000} C_DIS
LIN {X -162.631,Y -158.494,Z 160.000,A 0.000,B 0.000,C 180.000,E1 0.000} C_DIS
LIN {X -154.254,Y -166.657,Z 160.000,A 0.000,B 0.000,C 180.000,E1 0.000} C_DIS
LIN {X -145.471,Y -174.377,Z 160.000,A 0.000,B 0.000,C 180.000,E1 0.000} C_DIS
LIN {X -136.302,Y -181.634,Z 160.000,A 0.000,B 0.000,C 180.000,E1 0.000} C_DIS
LIN {X -126.770,Y -188.410,Z 160.000,A 0.000,B 0.000,C 180.000,E1 0.000} C_DIS
LIN {X -116.903,Y -194.686,Z 160.000,A 0.000,B 0.000,C 180.000,E1 0.000} C_DIS
LIN {X -106.726,Y -200.446,Z 160.000,A 0.000,B 0.000,C 180.000,E1 0.000} C_DIS
LIN {X -96.266,Y -205.675,Z 160.000,A 0.000,B 0.000,C 180.000,E1 0.000} C_DIS
LIN {X -85.547,Y -210.359,Z 160.000,A 0.000,B 0.000,C 180.000,E1 0.000} C_DIS
LIN {X -74.609,Y -214.483,Z 160.000,A 0.000,B 0.000,C 180.000,E1 0.000} C_DIS
LIN {X -63.468,Y -218.039,Z 160.000,A 0.000,B 0.000,C 180.000,E1 0.000} C_DIS
LIN {X -52.160,Y -221.018,Z 160.000,A 0.000,B 0.000,C 180.000,E1 0.000} C_DIS
LIN {X -40.713,Y -223.409,Z 160.000,A 0.000,B 0.000,C 180.000,E1 0.000} C_DIS
LIN {X -29.158,Y -225.209,Z 160.000,A 0.000,B 0.000,C 180.000,E1 0.000} C_DIS
LIN {X -17.525,Y -226.411,Z 160.000,A 0.000,B 0.000,C 180.000,E1 0.000} C_DIS
LIN {X -5.846,Y -227.013,Z 160.000,A 0.000,B 0.000,C 180.000,E1 0.000} C_DIS
LIN {X 5.846,Y -227.013,Z 160.000,A 0.000,B 0.000,C 180.000,E1 0.000} C_DIS
LIN {X 17.525,Y -226.411,Z 160.000,A 0.000,B 0.000,C 180.000,E1 0.000} C_DIS
LIN {X 29.158,Y -225.209,Z 160.000,A 0.000,B 0.000,C 180.000,E1 0.000} C_DIS
LIN {X 40.713,Y -223.409,Z 160.000,A 0.000,B 0.000,C 180.000,E1 0.000} C_DIS
LIN {X 52.160,Y -221.018,Z 160.000,A 0.000,B 0.000,C 180.000,E1 0.000} C_DIS
;rapid-leaky
$VEL.CP=0.3
LIN {X 185.292,Y -97.238,Z 160.000,A 0.000,B 0.000,C 180.000,E1 0.000} C_DIS
;bead-sparse_infill
$VEL.CP=0.62
LIN {X 97.154,Y -185.376,Z 160.000,A 0.000,B 0.000,C 180.000,E1 0.000} C_DIS
LIN {X 88.735,Y -189.584,Z 160.000,A 0.000,B 0.000,C 180.000,E1 0.000} C_DIS
LIN {X 78.858,Y -193.900,Z 160.000,A 0.000,B 0.000,C 180.000,E1 0.000} C_DIS
LIN {X 68.771,Y -197.703,Z 160.000,A 0.000,B 0.000,C 180.000,E1 0.000} C_DIS
LIN {X 58.502,Y -200.981,Z 160.000,A 0.000,B 0.000,C 180.000,E1 0.000} C_DIS
LIN {X 48.079,Y -203.727,Z 160.000,A 0.000,B 0.000,C 180.000,E1 0.000} C_DIS
LIN {X 37.528,Y -205.931,Z 160.000,A 0.000,B 0.000,C 180.000,E1 0.000} C_DIS
LIN {X 26.877,Y -207.590,Z 160.000,A 0.000,B 0.000,C 180.000,E1 0.000} C_DIS
LIN {X 16.154,Y -208.698,Z 160.000,A 0.000,B 0.000,C 180.000,E1 0.000} C_DIS
LIN {X 5.389,Y -209.253,Z 160.000,A 0.000,B 0.000,C 180.000,E1 0.000} C_DIS
LIN {X -5.389,Y -209.253,Z 160.000,A 0.000,B 0.000,C 180.000,E1 0.000} C_DIS
LIN {X -16.154,Y -208.698,Z 160.000,A 0.000,B 0.000,C 180.000,E1 0.000} C_DIS
LIN {X -26.877,Y -207.590,Z 160.000,A 0.000,B 0.000,C 180.000,E1 0.000} C_DIS
LIN {X -37.528,Y -205.931,Z 160.000,A 0.000,B 0.000,C 180.000,E1 0.000} C_DIS
LIN {X -48.079,Y -203.727,Z 160.000,A 0.000,B 0.000,C 180.000,E1 0.000} C_DIS
LIN {X -58.502,Y -200.981,Z 160.000,A 0.000,B 0.000,C 180.000,E1 0.000} C_DIS
LIN {X -68.772,Y -197.703,Z 160.000,A 0.000,B 0.000,C 180.000,E1 0.000} C_DIS
LIN {X -71.226,Y -196.778,Z 160.000,A 0.000,B 0.000,C 180.000,E1 0.000} C_DIS
LIN {X 196.776,Y 71.224,Z 160.000,A 0.000,B 0.000,C 180.000,E1 0.000} C_DIS
LIN {X 195.867,Y 73.837,Z 160.000,A 0.000,B 0.000,C 180.000,E1 0.000} C_DIS
LIN {X 191.804,Y 83.827,Z 160.000,A 0.000,B 0.000,C 180.000,E1 0.000} C_DIS
LIN {X 187.236,Y 93.587,Z 160.000,A 0.000,B 0.000,C 180.000,E1 0.000} C_DIS
LIN {X 182.169,Y 103.103,Z 160.000,A 0.000,B 0.000,C 180.000,E1 0.000} C_DIS
LIN {X 176.622,Y 112.343,Z 160.000,A 0.000,B 0.000,C 180.000,E1 0.000} C_DIS
LIN {X 170.604,Y 121.286,Z 160.000,A 0.000,B 0.000,C 180.000,E1 0.000} C_DIS
LIN {X 164.135,Y 129.907,Z 160.000,A 0.000,B 0.000,C 180.000,E1 0.000} C_DIS
LIN {X 157.229,Y 138.184,Z 160.000,A 0.000,B 0.000,C 180.000,E1 0.000} C_DIS
LIN {X 149.908,Y 146.094,Z 160.000,A 0.000,B 0.000,C 180.000,E1 0.000} C_DIS
LIN {X 142.186,Y 153.619,Z 160.000,A 0.000,B 0.000,C 180.000,E1 0.000} C_DIS
LIN {X 134.090,Y 160.736,Z 160.000,A 0.000,B 0.000,C 180.000,E1 0.000} C_DIS
LIN {X 131.422,Y 162.848,Z 160.000,A 0.000,B 0.000,C 180.000,E1 0.000} C_DIS
LIN {X -162.860,Y -131.435,Z 160.000,A 0.000,B 0.000,C 180.000,E1 0.000} C_DIS
LIN {X -164.135,Y -129.907,Z 160.000,A 0.000,B 0.000,C 180.000,E1 0.000} C_DIS
LIN {X -170.604,Y -121.286,Z 160.000,A 0.000,B 0.000,C 180.000,E1 0.000} C_DIS
